LIN {X 0,Y 579.036,Z 911.007,A -85,B 0,C 180,E1 18401.072,E2 18401.072} C_VEL
LIN {X 0,Y 580.6,Z 886.113,A -85,B 0,C 180,E1 18400.644,E2 18400.644} C_VEL
LIN {X 0,Y 588.894,Z 664.984,A -85,B 0,C 180,E1 18397.408,E2 18397.408} C_VEL
LIN {X 0,Y 594.592,Z 519.024,A -85,B 0,C 180,E1 18395.226,E2 18395.226} C_VEL
LIN {X 0,Y 583.238,Z 502.183,A -85,B 0,C 180,E1 18393.242,E2 18393.242} C_VEL
LIN {X 0,Y 573.346,Z 488.224,A -85,B 0,C 180,E1 18391.371,E2 18391.371} C_VEL
LIN {X 0,Y 562.808,Z 474.786,A -85,B 0,C 180,E1 18389.217,E2 18389.217} C_VEL
LIN {X 0,Y 557.617,Z 468.552,A -85,B 0,C 180,E1 18388.08,E2 18388.08} C_VEL
LIN {X 0,Y 553.132,Z 463.086,A -85,B 0,C 180,E1 18387.042,E2 18387.042} C_VEL
LIN {X 0,Y 548.609,Z 457.659,A -85,B 0,C 180,E1 18385.94,E2 18385.94} C_VEL
LIN {X 0,Y 544.992,Z 453.494,A -85,B 0,C 180,E1 18385.018,E2 18385.018} C_VEL
LIN {X 0,Y 543.71,Z 451.828,A -85,B 0,C 180,E1 18384.674,E2 18384.674} C_VEL
LIN {X 0,Y 540.306,Z 448.41,A -85,B 0,C 180,E1 18383.764,E2 18383.764} C_VEL
LIN {X 0,Y 538.516,Z 445.758,A -85,B 0,C 180,E1 18383.239,E2 18383.239} C_VEL
LIN {X 0,Y 535.176,Z 442.868,A -85,B 0,C 180,E1 18382.289,E2 18382.289} C_VEL
LIN {X 0,Y 532.967,Z 439.362,A -85,B 0,C 180,E1 18381.575,E2 18381.575} C_VEL
LIN {X 0,Y 529.819,Z 437.07,A -85,B 0,C 180,E1 18380.608,E2 18380.608} C_VEL
LIN {X 0,Y 527.865,Z 433.796,A -85,B 0,C 180,E1 18379.907,E2 18379.907} C_VEL
LIN {X 0,Y 527.382,Z 432.859,A -85,B 0,C 180,E1 18379.723,E2 18379.723} C_VEL
LIN {X 0,Y 524.15,Z 431.063,A -85,B 0,C 180,E1 18378.635,E2 18378.635} C_VEL
LIN {X 0,Y 522.344,Z 428.45,A -85,B 0,C 180,E1 18377.922,E2 18377.922} C_VEL
LIN {X 0,Y 521.734,Z 426.245,A -85,B 0,C 180,E1 18377.569,E2 18377.569} C_VEL
LIN {X 0,Y 521.677,Z 426.183,A -85,B 0,C 180,E1 18374.315,E2 18374.315} C_VEL
LIN {X 0,Y 521.681,Z 426.216,A -85,B 0,C 180,E1 18370.826,E2 18370.826} C_VEL
LIN {X 0,Y 521.736,Z 426.191,A -85,B 0,C 180,E1 18367.488,E2 18367.488} C_VEL
LIN {X 0,Y 521.667,Z 426.198,A -85,B 0,C 180,E1 18364.177,E2 18364.177} C_VEL
LIN {X 0,Y 521.698,Z 426.217,A -85,B 0,C 180,E1 18360.769,E2 18360.769} C_VEL
LIN {X 0,Y 521.675,Z 426.189,A -85,B 0,C 180,E1 18357.693,E2 18357.693} C_VEL
LIN {X 0,Y 521.674,Z 426.24,A -85,B 0,C 180,E1 18354.17,E2 18354.17} C_VEL
LIN {X 0,Y 521.705,Z 426.178,A -85,B 0,C 180,E1 18351.069,E2 18351.069} C_VEL
LIN {X 0,Y 521.667,Z 426.25,A -85,B 0,C 180,E1 18347.716,E2 18347.716} C_VEL
LIN {X 0,Y 521.718,Z 426.177,A -85,B 0,C 180,E1 18344.436,E2 18344.436} C_VEL
LIN {X 0,Y 521.761,Z 426.459,A -85,B 0,C 180,E1 18342.476,E2 18342.476} C_VEL
LIN {X 0,Y 522.696,Z 429.249,A -85,B 0,C 180,E1 18342.033,E2 18342.033} C_VEL
LIN {X 0,Y 525.013,Z 431.775,A -85,B 0,C 180,E1 18341.167,E2 18341.167} C_VEL
LIN {X 0,Y 527.588,Z 433.099,A -85,B 0,C 180,E1 18340.313,E2 18340.313} C_VEL
LIN {X 0,Y 529.339,Z 436.508,A -85,B 0,C 180,E1 18339.661,E2 18339.661} C_VEL
LIN {X 0,Y 532.257,Z 439.002,A -85,B 0,C 180,E1 18338.742,E2 18338.742} C_VEL
LIN {X 0,Y 533.358,Z 439.775,A -85,B 0,C 180,E1 18338.413,E2 18338.413} C_VEL
LIN {X 0,Y 535.655,Z 443.463,A -85,B 0,C 180,E1 18337.674,E2 18337.674} C_VEL
LIN {X 0,Y 539.017,Z 446.356,A -85,B 0,C 180,E1 18336.726,E2 18336.726} C_VEL
LIN {X 0,Y 541.984,Z 450.42,A -85,B 0,C 180,E1 18335.881,E2 18335.881} C_VEL
LIN {X 0,Y 544.316,Z 452.723,A -85,B 0,C 180,E1 18335.268,E2 18335.268} C_VEL
LIN {X 0,Y 552.544,Z 463.032,A -85,B 0,C 180,E1 18333.189,E2 18333.189} C_VEL
LIN {X 0,Y 558.316,Z 470.524,A -85,B 0,C 180,E1 18331.842,E2 18331.842} C_VEL
LIN {X 0,Y 566.802,Z 481.647,A -85,B 0,C 180,E1 18330.006,E2 18330.006} C_VEL
LIN {X 0,Y 579.311,Z 499.123,A -85,B 0,C 180,E1 18327.535,E2 18327.535} C_VEL
LIN {X 0,Y 591.797,Z 517.896,A -85,B 0,C 180,E1 18325.292,E2 18325.292} C_VEL
LIN {X 0,Y 594.718,Z 522.57,A -85,B 0,C 180,E1 18324.793,E2 18324.793} C_VEL
LIN {X 0,Y 586.211,Z 739.964,A -85,B 0,C 180,E1 18321.576,E2 18321.576} C_VEL
LIN {X 0,Y 580.04,Z 903.137,A -85,B 0,C 180,E1 18319.182,E2 18319.182} C_VEL
LIN {X 0,Y 578.241,Z 928.181,A -85,B 0,C 180,E1 18318.717,E2 18318.717} C_VEL
LIN {X 0,Y 575.436,Z 956.17,A -85,B 0,C 180,E1 18318.007,E2 18318.007} C_VEL
LIN {X 0,Y 572.745,Z 978.261,A -85,B 0,C 180,E1 18317.298,E2 18317.298} C_VEL
LIN {X 0,Y 569.876,Z 998.966,A -85,B 0,C 180,E1 18316.505,E2 18316.505} C_VEL
LIN {X 0,Y 566.742,Z 1019.265,A -85,B 0,C 180,E1 18315.598,E2 18315.598} C_VEL
LIN {X 0,Y 562.552,Z 1044.182,A -85,B 0,C 180,E1 18314.302,E2 18314.302} C_VEL
LIN {X 0,Y 558.22,Z 1067.089,A -85,B 0,C 180,E1 18312.889,E2 18312.889} C_VEL
LIN {X 0,Y 554.385,Z 1086.314,A -85,B 0,C 180,E1 18311.539,E2 18311.539} C_VEL
LIN {X 0,Y 550.54,Z 1104.879,A -85,B 0,C 180,E1 18310.073,E2 18310.073} C_VEL
LIN {X 0,Y 546.407,Z 1124.422,A -85,B 0,C 180,E1 18308.335,E2 18308.335} C_VEL
LIN {X 0,Y 541.6,Z 1146.573,A -85,B 0,C 180,E1 18306.075,E2 18306.075} C_VEL
LIN {X 0,Y 538.12,Z 1162.602,A -85,B 0,C 180,E1 18304.222,E2 18304.222} C_VEL
LIN {X 0,Y 534.941,Z 1177.486,A -85,B 0,C 180,E1 18302.31,E2 18302.31} C_VEL
LIN {X 0,Y 532.102,Z 1191.164,A -85,B 0,C 180,E1 18300.358,E2 18300.358} C_VEL
LIN {X 0,Y 528.99,Z 1207.163,A -85,B 0,C 180,E1 18297.796,E2 18297.796} C_VEL
LIN {X 0,Y 526.229,Z 1221.856,A -85,B 0,C 180,E1 18295.065,E2 18295.065} C_VEL
LIN {X 0,Y 524.427,Z 1232.786,A -85,B 0,C 180,E1 18292.766,E2 18292.766} C_VEL
LIN {X 0,Y 522.967,Z 1242.909,A -85,B 0,C 180,E1 18290.359,E2 18290.359} C_VEL
LIN {X 0,Y 521.584,Z 1254.042,A -85,B 0,C 180,E1 18287.282,E2 18287.282} C_VEL
LIN {X 0,Y 520.803,Z 1261.844,A -85,B 0,C 180,E1 18284.676,E2 18284.676} C_VEL
LIN {X 0,Y 520.369,Z 1267.807,A -85,B 0,C 180,E1 18282.311,E2 18282.311} C_VEL
LIN {X 0,Y 520.093,Z 1272.702,A -85,B 0,C 180,E1 18279.96,E2 18279.96} C_VEL
LIN {X 0,Y 519.964,Z 1276.525,A -85,B 0,C 180,E1 18277.621,E2 18277.621} C_VEL
LIN {X 0,Y 519.925,Z 1279.433,A -85,B 0,C 180,E1 18275.182,E2 18275.182} C_VEL
LIN {X 0,Y 519.907,Z 1281.491,A -85,B 0,C 180,E1 18272.311,E2 18272.311} C_VEL
LIN {X 0,Y 519.867,Z 1281.893,A -85,B 0,C 180,E1 18269.446,E2 18269.446} C_VEL
LIN {X 0,Y 519.91,Z 1281.08,A -85,B 0,C 180,E1 18267.02,E2 18267.02} C_VEL
LIN {X 0,Y 519.926,Z 1279.198,A -85,B 0,C 180,E1 18264.59,E2 18264.59} C_VEL
LIN {X 0,Y 519.965,Z 1276.355,A -85,B 0,C 180,E1 18262.261,E2 18262.261} C_VEL
LIN {X 0,Y 520.127,Z 1272.277,A -85,B 0,C 180,E1 18259.81,E2 18259.81} C_VEL
LIN {X 0,Y 520.467,Z 1266.52,A -85,B 0,C 180,E1 18257.121,E2 18257.121} C_VEL
LIN {X 0,Y 521.149,Z 1258.259,A -85,B 0,C 180,E1 18254.073,E2 18254.073} C_VEL
LIN {X 0,Y 522.037,Z 1250.093,A -85,B 0,C 180,E1 18251.574,E2 18251.574} C_VEL
LIN {X 0,Y 523.226,Z 1241.051,A -85,B 0,C 180,E1 18249.177,E2 18249.177} C_VEL
LIN {X 0,Y 524.865,Z 1230.188,A -85,B 0,C 180,E1 18246.654,E2 18246.654} C_VEL
LIN {X 0,Y 527.442,Z 1215.245,A -85,B 0,C 180,E1 18243.664,E2 18243.664} C_VEL
LIN {X 0,Y 529.901,Z 1202.05,A -85,B 0,C 180,E1 18241.359,E2 18241.359} C_VEL
LIN {X 0,Y 532.597,Z 1188.807,A -85,B 0,C 180,E1 18239.291,E2 18239.291} C_VEL
LIN {X 0,Y 535.704,Z 1174.039,A -85,B 0,C 180,E1 18237.227,E2 18237.227} C_VEL
LIN {X 0,Y 540.173,Z 1153.102,A -85,B 0,C 180,E1 18234.652,E2 18234.652} C_VEL
LIN {X 0,Y 543.91,Z 1135.76,A -85,B 0,C 180,E1 18232.783,E2 18232.783} C_VEL
LIN {X 0,Y 547.556,Z 1118.85,A -85,B 0,C 180,E1 18231.15,E2 18231.15} C_VEL
LIN {X 0,Y 551.544,Z 1100.101,A -85,B 0,C 180,E1 18229.531,E2 18229.531} C_VEL
LIN {X 0,Y 556.662,Z 1075.128,A -85,B 0,C 180,E1 18227.654,E2 18227.654} C_VEL
LIN {X 0,Y 560.526,Z 1054.925,A -85,B 0,C 180,E1 18226.341,E2 18226.341} C_VEL
LIN {X 0,Y 563.912,Z 1036.027,A -85,B 0,C 180,E1 18225.255,E2 18225.255} C_VEL
LIN {X 0,Y 567.295,Z 1015.734,A -85,B 0,C 180,E1 18224.234,E2 18224.234} C_VEL
LIN {X 0,Y 570.571,Z 994.236,A -85,B 0,C 180,E1 18223.301,E2 18223.301} C_VEL
LIN {X 0,Y 574.261,Z 966.352,A -85,B 0,C 180,E1 18222.3,E2 18222.3} C_VEL
LIN {X 0,Y 576.846,Z 942.712,A -85,B 0,C 180,E1 18221.629,E2 18221.629} C_VEL
LIN {X 0,Y 578.774,Z 921.217,A -85,B 0,C 180,E1 18221.143,E2 18221.143} C_VEL
LIN {X 0,Y 580.258,Z 898.846,A -85,B 0,C 180,E1 18220.75,E2 18220.75} C_VEL
LIN {X 0,Y 588.488,Z 679.578,A -85,B 0,C 180,E1 18217.538,E2 18217.538} C_VEL
LIN {X 0,Y 594.641,Z 522.279,A -85,B 0,C 180,E1 18215.196,E2 18215.196} C_VEL
LIN {X 0,Y 582.085,Z 503.302,A -85,B 0,C 180,E1 18212.993,E2 18212.993} C_VEL
LIN {X 0,Y 571.124,Z 487.581,A -85,B 0,C 180,E1 18210.891,E2 18210.891} C_VEL
LIN {X 0,Y 559.93,Z 472.501,A -85,B 0,C 180,E1 18208.535,E2 18208.535} C_VEL
LIN {X 0,Y 554.757,Z 466.005,A -85,B 0,C 180,E1 18207.362,E2 18207.362} C_VEL
LIN {X 0,Y 550.787,Z 460.835,A -85,B 0,C 180,E1 18206.409,E2 18206.409} C_VEL
LIN {X 0,Y 543.204,Z 451.467,A -85,B 0,C 180,E1 18204.467,E2 18204.467} C_VEL
LIN {X 0,Y 539.929,Z 447.877,A -85,B 0,C 180,E1 18203.579,E2 18203.579} C_VEL
LIN {X 0,Y 538.57,Z 445.796,A -85,B 0,C 180,E1 18203.178,E2 18203.178} C_VEL
LIN {X 0,Y 535.297,Z 443.031,A -85,B 0,C 180,E1 18202.255,E2 18202.255} C_VEL
LIN {X 0,Y 533.175,Z 439.455,A -85,B 0,C 180,E1 18201.566,E2 18201.566} C_VEL
LIN {X 0,Y 529.837,Z 437.087,A -85,B 0,C 180,E1 18200.549,E2 18200.549} C_VEL
LIN {X 0,Y 527.874,Z 433.805,A -85,B 0,C 180,E1 18199.848,E2 18199.848} C_VEL
LIN {X 0,Y 527.553,Z 432.909,A -85,B 0,C 180,E1 18199.717,E2 18199.717} C_VEL
LIN {X 0,Y 524.143,Z 431.05,A -85,B 0,C 180,E1 18198.577,E2 18198.577} C_VEL
LIN {X 0,Y 522.271,Z 428.25,A -85,B 0,C 180,E1 18197.838,E2 18197.838} C_VEL
LIN {X 0,Y 521.734,Z 426.244,A -85,B 0,C 180,E1 18197.54,E2 18197.54} C_VEL
LIN {X 0,Y 521.706,Z 426.183,A -85,B 0,C 180,E1 18194.201,E2 18194.201} C_VEL
LIN {X 0,Y 521.699,Z 426.209,A -85,B 0,C 180,E1 18190.826,E2 18190.826} C_VEL
LIN {X 0,Y 521.751,Z 426.198,A -85,B 0,C 180,E1 18187.377,E2 18187.377} C_VEL
LIN {X 0,Y 521.711,Z 426.185,A -85,B 0,C 180,E1 18184.066,E2 18184.066} C_VEL
LIN {X 0,Y 521.713,Z 426.233,A -85,B 0,C 180,E1 18180.549,E2 18180.549} C_VEL
LIN {X 0,Y 521.737,Z 426.171,A -85,B 0,C 180,E1 18177.144,E2 18177.144} C_VEL
LIN {X 0,Y 521.743,Z 426.239,A -85,B 0,C 180,E1 18173.618,E2 18173.618} C_VEL
LIN {X 0,Y 521.718,Z 426.181,A -85,B 0,C 180,E1 18170.099,E2 18170.099} C_VEL
LIN {X 0,Y 521.743,Z 426.202,A -85,B 0,C 180,E1 18166.704,E2 18166.704} C_VEL
LIN {X 0,Y 521.738,Z 426.209,A -85,B 0,C 180,E1 18163.179,E2 18163.179} C_VEL
LIN {X 0,Y 521.765,Z 426.425,A -85,B 0,C 180,E1 18162.216,E2 18162.216} C_VEL
LIN {X 0,Y 522.647,Z 429.071,A -85,B 0,C 180,E1 18161.801,E2 18161.801} C_VEL
LIN {X 0,Y 525.115,Z 431.787,A -85,B 0,C 180,E1 18160.882,E2 18160.882} C_VEL
LIN {X 0,Y 527.676,Z 433.195,A -85,B 0,C 180,E1 18160.036,E2 18160.036} C_VEL
LIN {X 0,Y 529.467,Z 436.573,A -85,B 0,C 180,E1 18159.378,E2 18159.378} C_VEL
LIN {X 0,Y 532.576,Z 439.16,A -85,B 0,C 180,E1 18158.409,E2 18158.409} C_VEL
LIN {X 0,Y 533.5,Z 439.944,A -85,B 0,C 180,E1 18158.13,E2 18158.13} C_VEL
LIN {X 0,Y 535.819,Z 443.573,A -85,B 0,C 180,E1 18157.392,E2 18157.392} C_VEL
LIN {X 0,Y 539.108,Z 446.411,A -85,B 0,C 180,E1 18156.47,E2 18156.47} C_VEL
LIN {X 0,Y 541.999,Z 450.36,A -85,B 0,C 180,E1 18155.649,E2 18155.649} C_VEL
LIN {X 0,Y 544.45,Z 452.616,A -85,B 0,C 180,E1 18155.014,E2 18155.014} C_VEL
LIN {X 0,Y 547.821,Z 456.922,A -85,B 0,C 180,E1 18154.137,E2 18154.137} C_VEL
LIN {X 0,Y 549.689,Z 458.859,A -85,B 0,C 180,E1 18153.68,E2 18153.68} C_VEL
LIN {X 0,Y 553.558,Z 463.505,A -85,B 0,C 180,E1 18152.748,E2 18152.748} C_VEL
LIN {X 0,Y 559.954,Z 471.36,A -85,B 0,C 180,E1 18151.292,E2 18151.292} C_VEL
LIN {X 0,Y 568.098,Z 481.467,A -85,B 0,C 180,E1 18149.572,E2 18149.572} C_VEL
LIN {X 0,Y 576.042,Z 491.922,A -85,B 0,C 180,E1 18148.004,E2 18148.004} C_VEL
LIN {X 0,Y 588.387,Z 509.679,A -85,B 0,C 180,E1 18145.742,E2 18145.742} C_VEL
LIN {X 0,Y 594.647,Z 519.437,A -85,B 0,C 180,E1 18144.662,E2 18144.662} C_VEL
LIN {X 0,Y 586.266,Z 733.251,A -85,B 0,C 180,E1 18141.497,E2 18141.497} C_VEL
LIN {X 0,Y 580.128,Z 894.828,A -85,B 0,C 180,E1 18139.126,E2 18139.126} C_VEL
LIN {X 0,Y 578.382,Z 919.425,A -85,B 0,C 180,E1 18138.667,E2 18138.667} C_VEL
LIN {X 0,Y 575.597,Z 947.533,A -85,B 0,C 180,E1 18137.952,E2 18137.952} C_VEL
LIN {X 0,Y 573.377,Z 966.175,A -85,B 0,C 180,E1 18137.362,E2 18137.362} C_VEL
LIN {X 0,Y 571.693,Z 973.633,A -85,B 0,C 180,E1 18137.174,E2 18137.174} C_VEL
LIN {X 0,Y 564.929,Z 992.335,A -85,B 0,C 180,E1 18136.894,E2 18136.894} C_VEL
LIN {X 0,Y 563.145,Z 999.439,A -85,B 0,C 180,E1 18136.66,E2 18136.66} C_VEL
LIN {X 0,Y 558.919,Z 1024.068,A -85,B 0,C 180,E1 18135.448,E2 18135.448} C_VEL
LIN {X 0,Y 555.437,Z 1042.82,A -85,B 0,C 180,E1 18134.383,E2 18134.383} C_VEL
LIN {X 0,Y 551.84,Z 1060.85,A -85,B 0,C 180,E1 18133.23,E2 18133.23} C_VEL
LIN {X 0,Y 547.962,Z 1079.276,A -85,B 0,C 180,E1 18131.903,E2 18131.903} C_VEL
LIN {X 0,Y 543.746,Z 1098.556,A -85,B 0,C 180,E1 18130.339,E2 18130.339} C_VEL
LIN {X 0,Y 538.534,Z 1121.584,A -85,B 0,C 180,E1 18128.192,E2 18128.192} C_VEL
LIN {X 0,Y 534.458,Z 1139.111,A -85,B 0,C 180,E1 18126.322,E2 18126.322} C_VEL
LIN {X 0,Y 530.92,Z 1154.438,A -85,B 0,C 180,E1 18124.496,E2 18124.496} C_VEL
LIN {X 0,Y 527.405,Z 1169.864,A -85,B 0,C 180,E1 18122.45,E2 18122.45} C_VEL
LIN {X 0,Y 523.546,Z 1187.627,A -85,B 0,C 180,E1 18119.775,E2 18119.775} C_VEL
LIN {X 0,Y 520.587,Z 1201.836,A -85,B 0,C 180,E1 18117.328,E2 18117.328} C_VEL
LIN {X 0,Y 518.387,Z 1213.335,A -85,B 0,C 180,E1 18115.111,E2 18115.111} C_VEL
LIN {X 0,Y 516.527,Z 1224.112,A -85,B 0,C 180,E1 18112.78,E2 18112.78} C_VEL
LIN {X 0,Y 514.77,Z 1235.881,A -85,B 0,C 180,E1 18109.874,E2 18109.874} C_VEL
LIN {X 0,Y 513.521,Z 1245.65,A -85,B 0,C 180,E1 18106.984,E2 18106.984} C_VEL
LIN {X 0,Y 512.833,Z 1252.312,A -85,B 0,C 180,E1 18104.685,E2 18104.685} C_VEL
LIN {X 0,Y 512.394,Z 1257.946,A -85,B 0,C 180,E1 18102.398,E2 18102.398} C_VEL
LIN {X 0,Y 512.109,Z 1262.812,A -85,B 0,C 180,E1 18100.01,E2 18100.01} C_VEL
LIN {X 0,Y 511.962,Z 1266.768,A -85,B 0,C 180,E1 18097.522,E2 18097.522} C_VEL
LIN {X 0,Y 511.921,Z 1269.832,A -85,B 0,C 180,E1 18094.821,E2 18094.821} C_VEL
LIN {X 0,Y 511.908,Z 1271.634,A -85,B 0,C 180,E1 18091.794,E2 18091.794} C_VEL
LIN {X 0,Y 511.865,Z 1271.858,A -85,B 0,C 180,E1 18089.22,E2 18089.22} C_VEL
LIN {X 0,Y 511.911,Z 1271.043,A -85,B 0,C 180,E1 18086.868,E2 18086.868} C_VEL
LIN {X 0,Y 511.928,Z 1269.249,A -85,B 0,C 180,E1 18084.512,E2 18084.512} C_VEL
LIN {X 0,Y 511.973,Z 1266.426,A -85,B 0,C 180,E1 18082.146,E2 18082.146} C_VEL
LIN {X 0,Y 512.147,Z 1262.368,A -85,B 0,C 180,E1 18079.656,E2 18079.656} C_VEL
LIN {X 0,Y 512.511,Z 1256.635,A -85,B 0,C 180,E1 18076.924,E2 18076.924} C_VEL
LIN {X 0,Y 513.225,Z 1248.418,A -85,B 0,C 180,E1 18073.828,E2 18073.828} C_VEL
LIN {X 0,Y 514.17,Z 1240.216,A -85,B 0,C 180,E1 18071.273,E2 18071.273} C_VEL
LIN {X 0,Y 515.427,Z 1231.245,A -85,B 0,C 180,E1 18068.854,E2 18068.854} C_VEL
LIN {X 0,Y 517.076,Z 1220.916,A -85,B 0,C 180,E1 18066.409,E2 18066.409} C_VEL
LIN {X 0,Y 519.684,Z 1206.642,A -85,B 0,C 180,E1 18063.467,E2 18063.467} C_VEL
LIN {X 0,Y 522.37,Z 1192.914,A -85,B 0,C 180,E1 18061.018,E2 18061.018} C_VEL
LIN {X 0,Y 525.169,Z 1179.971,A -85,B 0,C 180,E1 18058.943,E2 18058.943} C_VEL
LIN {X 0,Y 528.229,Z 1166.296,A -85,B 0,C 180,E1 18056.97,E2 18056.97} C_VEL
LIN {X 0,Y 531.991,Z 1149.884,A -85,B 0,C 180,E1 18054.845,E2 18054.845} C_VEL
LIN {X 0,Y 536.787,Z 1129.016,A -85,B 0,C 180,E1 18052.481,E2 18052.481} C_VEL
LIN {X 0,Y 540.792,Z 1111.502,A -85,B 0,C 180,E1 18050.739,E2 18050.739} C_VEL
LIN {X 0,Y 544.691,Z 1094.186,A -85,B 0,C 180,E1 18049.2,E2 18049.2} C_VEL
LIN {X 0,Y 548.793,Z 1075.37,A -85,B 0,C 180,E1 18047.708,E2 18047.708} C_VEL
LIN {X 0,Y 553.8,Z 1051.295,A -85,B 0,C 180,E1 18046.042,E2 18046.042} C_VEL
LIN {X 0,Y 557.992,Z 1029.086,A -85,B 0,C 180,E1 18044.731,E2 18044.731} C_VEL
LIN {X 0,Y 561.497,Z 1009.094,A -85,B 0,C 180,E1 18043.704,E2 18043.704} C_VEL
LIN {X 0,Y 564.561,Z 989.967,A -85,B 0,C 180,E1 18042.849,E2 18042.849} C_VEL
LIN {X 0,Y 567.434,Z 969.925,A -85,B 0,C 180,E1 18042.076,E2 18042.076} C_VEL
LIN {X 0,Y 570.195,Z 947.979,A -85,B 0,C 180,E1 18041.366,E2 18041.366} C_VEL
LIN {X 0,Y 573.055,Z 920.319,A -85,B 0,C 180,E1 18040.655,E2 18040.655} C_VEL
LIN {X 0,Y 574.916,Z 895.077,A -85,B 0,C 180,E1 18040.181,E2 18040.181} C_VEL
LIN {X 0,Y 580.74,Z 748.236,A -85,B 0,C 180,E1 18038.012,E2 18038.012} C_VEL
LIN {X 0,Y 589.427,Z 534.986,A -85,B 0,C 180,E1 18034.843,E2 18034.843} C_VEL
LIN {X 0,Y 589.825,Z 523.275,A -85,B 0,C 180,E1 18034.653,E2 18034.653} C_VEL
LIN {X 0,Y 579.401,Z 507.75,A -85,B 0,C 180,E1 18032.782,E2 18032.782} C_VEL
LIN {X 0,Y 569.991,Z 494.34,A -85,B 0,C 180,E1 18030.959,E2 18030.959} C_VEL
LIN {X 0,Y 559.803,Z 481.353,A -85,B 0,C 180,E1 18028.833,E2 18028.833} C_VEL
LIN {X 0,Y 554.789,Z 475.248,A -85,B 0,C 180,E1 18027.71,E2 18027.71} C_VEL
LIN {X 0,Y 550.666,Z 470.149,A -85,B 0,C 180,E1 18026.735,E2 18026.735} C_VEL
LIN {X 0,Y 546.293,Z 464.859,A -85,B 0,C 180,E1 18025.65,E2 18025.65} C_VEL
LIN {X 0,Y 542.548,Z 460.371,A -85,B 0,C 180,E1 18024.672,E2 18024.672} C_VEL
LIN {X 0,Y 541.071,Z 458.796,A -85,B 0,C 180,E1 18024.279,E2 18024.279} C_VEL
LIN {X 0,Y 537.596,Z 454.789,A -85,B 0,C 180,E1 18023.31,E2 18023.31} C_VEL
LIN {X 0,Y 536.497,Z 453.235,A -85,B 0,C 180,E1 18022.983,E2 18022.983} C_VEL
LIN {X 0,Y 533.047,Z 450.017,A -85,B 0,C 180,E1 18021.976,E2 18021.976} C_VEL
LIN {X 0,Y 531.01,Z 446.911,A -85,B 0,C 180,E1 18021.31,E2 18021.31} C_VEL
LIN {X 0,Y 527.773,Z 444.256,A -85,B 0,C 180,E1 18020.286,E2 18020.286} C_VEL
LIN {X 0,Y 525.492,Z 440.526,A -85,B 0,C 180,E1 18019.45,E2 18019.45} C_VEL
LIN {X 0,Y 522.199,Z 438.327,A -85,B 0,C 180,E1 18018.302,E2 18018.302} C_VEL
LIN {X 0,Y 520.267,Z 435.183,A -85,B 0,C 180,E1 18017.504,E2 18017.504} C_VEL
LIN {X 0,Y 519.808,Z 434.015,A -85,B 0,C 180,E1 18017.289,E2 18017.289} C_VEL
LIN {X 0,Y 516.455,Z 432.216,A -85,B 0,C 180,E1 18015.957,E2 18015.957} C_VEL
LIN {X 0,Y 514.286,Z 429.246,A -85,B 0,C 180,E1 18014.928,E2 18014.928} C_VEL
LIN {X 0,Y 513.731,Z 427.169,A -85,B 0,C 180,E1 18014.541,E2 18014.541} C_VEL
LIN {X 0,Y 513.765,Z 427.211,A -85,B 0,C 180,E1 18011.109,E2 18011.109} C_VEL
LIN {X 0,Y 513.757,Z 427.174,A -85,B 0,C 180,E1 18007.83,E2 18007.83} C_VEL
LIN {X 0,Y 513.733,Z 427.192,A -85,B 0,C 180,E1 18004.465,E2 18004.465} C_VEL
LIN {X 0,Y 513.796,Z 427.185,A -85,B 0,C 180,E1 18001.115,E2 18001.115} C_VEL
LIN {X 0,Y 513.728,Z 427.18,A -85,B 0,C 180,E1 17997.881,E2 17997.881} C_VEL
LIN {X 0,Y 513.748,Z 427.214,A -85,B 0,C 180,E1 17994.415,E2 17994.415} C_VEL
LIN {X 0,Y 513.742,Z 427.17,A -85,B 0,C 180,E1 17991.344,E2 17991.344} C_VEL
LIN {X 0,Y 513.731,Z 427.239,A -85,B 0,C 180,E1 17987.866,E2 17987.866} C_VEL
LIN {X 0,Y 513.739,Z 427.322,A -85,B 0,C 180,E1 17985.517,E2 17985.517} C_VEL
LIN {X 0,Y 514.585,Z 429.867,A -85,B 0,C 180,E1 17985.023,E2 17985.023} C_VEL
LIN {X 0,Y 517.197,Z 432.829,A -85,B 0,C 180,E1 17983.836,E2 17983.836} C_VEL
LIN {X 0,Y 519.913,Z 434.245,A -85,B 0,C 180,E1 17982.772,E2 17982.772} C_VEL
LIN {X 0,Y 521.498,Z 437.521,A -85,B 0,C 180,E1 17982.077,E2 17982.077} C_VEL
LIN {X 0,Y 524.383,Z 440.031,A -85,B 0,C 180,E1 17981.026,E2 17981.026} C_VEL
LIN {X 0,Y 525.766,Z 440.869,A -85,B 0,C 180,E1 17980.56,E2 17980.56} C_VEL
LIN {X 0,Y 527.906,Z 444.43,A -85,B 0,C 180,E1 17979.777,E2 17979.777} C_VEL
LIN {X 0,Y 531.473,Z 447.447,A -85,B 0,C 180,E1 17978.651,E2 17978.651} C_VEL
LIN {X 0,Y 534.186,Z 451.376,A -85,B 0,C 180,E1 17977.784,E2 17977.784} C_VEL
LIN {X 0,Y 536.992,Z 453.833,A -85,B 0,C 180,E1 17976.982,E2 17976.982} C_VEL
LIN {X 0,Y 540.118,Z 457.965,A -85,B 0,C 180,E1 17976.082,E2 17976.082} C_VEL
LIN {X 0,Y 542.512,Z 460.465,A -85,B 0,C 180,E1 17975.442,E2 17975.442} C_VEL
LIN {X 0,Y 550.279,Z 470.345,A -85,B 0,C 180,E1 17973.449,E2 17973.449} C_VEL
LIN {X 0,Y 558.284,Z 480.701,A -85,B 0,C 180,E1 17971.578,E2 17971.578} C_VEL
LIN {X 0,Y 569.062,Z 495.522,A -85,B 0,C 180,E1 17969.278,E2 17969.278} C_VEL
LIN {X 0,Y 579.122,Z 510.073,A -85,B 0,C 180,E1 17967.317,E2 17967.317} C_VEL
LIN {X 0,Y 589.944,Z 526.608,A -85,B 0,C 180,E1 17965.369,E2 17965.369} C_VEL
LIN {X 0,Y 581.1,Z 743.647,A -85,B 0,C 180,E1 17962.142,E2 17962.142} C_VEL
LIN {X 0,Y 574.825,Z 902.956,A -85,B 0,C 180,E1 17959.79,E2 17959.79} C_VEL
LIN {X 0,Y 572.972,Z 927.943,A -85,B 0,C 180,E1 17959.326,E2 17959.326} C_VEL
LIN {X 0,Y 570.058,Z 956.08,A -85,B 0,C 180,E1 17958.611,E2 17958.611} C_VEL
LIN {X 0,Y 567.273,Z 978.178,A -85,B 0,C 180,E1 17957.9,E2 17957.9} C_VEL
LIN {X 0,Y 564.321,Z 998.754,A -85,B 0,C 180,E1 17957.11,E2 17957.11} C_VEL
LIN {X 0,Y 561.042,Z 1019.18,A -85,B 0,C 180,E1 17956.195,E2 17956.195} C_VEL
LIN {X 0,Y 556.686,Z 1044.095,A -85,B 0,C 180,E1 17954.894,E2 17954.894} C_VEL
LIN {X 0,Y 552.016,Z 1067.808,A -85,B 0,C 180,E1 17953.419,E2 17953.419} C_VEL
LIN {X 0,Y 547.988,Z 1087.181,A -85,B 0,C 180,E1 17952.043,E2 17952.043} C_VEL
LIN {X 0,Y 544.037,Z 1105.458,A -85,B 0,C 180,E1 17950.582,E2 17950.582} C_VEL
LIN {X 0,Y 539.227,Z 1127.368,A -85,B 0,C 180,E1 17948.601,E2 17948.601} C_VEL
LIN {X 0,Y 534.599,Z 1147.5,A -85,B 0,C 180,E1 17946.491,E2 17946.491} C_VEL
LIN {X 0,Y 530.982,Z 1163.398,A -85,B 0,C 180,E1 17944.622,E2 17944.622} C_VEL
LIN {X 0,Y 527.663,Z 1178.244,A -85,B 0,C 180,E1 17942.682,E2 17942.682} C_VEL
LIN {X 0,Y 524.012,Z 1195.317,A -85,B 0,C 180,E1 17940.186,E2 17940.186} C_VEL
LIN {X 0,Y 520.791,Z 1210.83,A -85,B 0,C 180,E1 17937.557,E2 17937.557} C_VEL
LIN {X 0,Y 518.462,Z 1222.903,A -85,B 0,C 180,E1 17935.243,E2 17935.243} C_VEL
LIN {X 0,Y 516.662,Z 1233.298,A -85,B 0,C 180,E1 17933.008,E2 17933.008} C_VEL
LIN {X 0,Y 514.998,Z 1244.284,A -85,B 0,C 180,E1 17930.332,E2 17930.332} C_VEL
LIN {X 0,Y 513.582,Z 1255.103,A -85,B 0,C 180,E1 17927.209,E2 17927.209} C_VEL
LIN {X 0,Y 512.836,Z 1262.276,A -85,B 0,C 180,E1 17924.745,E2 17924.745} C_VEL
LIN {X 0,Y 512.389,Z 1268.061,A -85,B 0,C 180,E1 17922.391,E2 17922.391} C_VEL
LIN {X 0,Y 512.102,Z 1272.906,A -85,B 0,C 180,E1 17920.004,E2 17920.004} C_VEL
LIN {X 0,Y 511.967,Z 1276.842,A -85,B 0,C 180,E1 17917.515,E2 17917.515} C_VEL
LIN {X 0,Y 511.92,Z 1279.996,A -85,B 0,C 180,E1 17914.702,E2 17914.702} C_VEL
LIN {X 0,Y 511.908,Z 1281.668,A -85,B 0,C 180,E1 17911.676,E2 17911.676} C_VEL
LIN {X 0,Y 511.866,Z 1281.848,A -85,B 0,C 180,E1 17909.213,E2 17909.213} C_VEL
LIN {X 0,Y 511.91,Z 1281.012,A -85,B 0,C 180,E1 17906.862,E2 17906.862} C_VEL
LIN {X 0,Y 511.929,Z 1279.196,A -85,B 0,C 180,E1 17904.505,E2 17904.505} C_VEL
LIN {X 0,Y 511.972,Z 1276.352,A -85,B 0,C 180,E1 17902.14,E2 17902.14} C_VEL
LIN {X 0,Y 512.156,Z 1272.274,A -85,B 0,C 180,E1 17899.65,E2 17899.65} C_VEL
LIN {X 0,Y 512.552,Z 1266.189,A -85,B 0,C 180,E1 17896.77,E2 17896.77} C_VEL
LIN {X 0,Y 513.279,Z 1257.905,A -85,B 0,C 180,E1 17893.706,E2 17893.706} C_VEL
LIN {X 0,Y 514.228,Z 1249.687,A -85,B 0,C 180,E1 17891.167,E2 17891.167} C_VEL
LIN {X 0,Y 515.457,Z 1241.049,A -85,B 0,C 180,E1 17888.848,E2 17888.848} C_VEL
LIN {X 0,Y 517.117,Z 1230.702,A -85,B 0,C 180,E1 17886.404,E2 17886.404} C_VEL
LIN {X 0,Y 519.82,Z 1215.878,A -85,B 0,C 180,E1 17883.371,E2 17883.371} C_VEL
LIN {X 0,Y 522.446,Z 1202.554,A -85,B 0,C 180,E1 17881.002,E2 17881.002} C_VEL
LIN {X 0,Y 525.214,Z 1189.501,A -85,B 0,C 180,E1 17878.939,E2 17878.939} C_VEL
LIN {X 0,Y 528.254,Z 1175.646,A -85,B 0,C 180,E1 17876.964,E2 17876.964} C_VEL
LIN {X 0,Y 532.349,Z 1157.54,A -85,B 0,C 180,E1 17874.653,E2 17874.653} C_VEL
LIN {X 0,Y 536.883,Z 1137.341,A -85,B 0,C 180,E1 17872.413,E2 17872.413} C_VEL
LIN {X 0,Y 540.798,Z 1119.98,A -85,B 0,C 180,E1 17870.708,E2 17870.708} C_VEL
LIN {X 0,Y 544.789,Z 1101.994,A -85,B 0,C 180,E1 17869.128,E2 17869.128} C_VEL
LIN {X 0,Y 549.427,Z 1080.555,A -85,B 0,C 180,E1 17867.46,E2 17867.46} C_VEL
LIN {X 0,Y 554.247,Z 1056.638,A -85,B 0,C 180,E1 17865.863,E2 17865.863} C_VEL
LIN {X 0,Y 557.931,Z 1036.941,A -85,B 0,C 180,E1 17864.716,E2 17864.716} C_VEL
LIN {X 0,Y 561.431,Z 1016.773,A -85,B 0,C 180,E1 17863.69,E2 17863.69} C_VEL
LIN {X 0,Y 564.515,Z 997.425,A -85,B 0,C 180,E1 17862.836,E2 17862.836} C_VEL
LIN {X 0,Y 567.565,Z 976.037,A -85,B 0,C 180,E1 17862.025,E2 17862.025} C_VEL
LIN {X 0,Y 570.859,Z 949.429,A -85,B 0,C 180,E1 17861.198,E2 17861.198} C_VEL
LIN {X 0,Y 573.306,Z 923.608,A -85,B 0,C 180,E1 17860.587,E2 17860.587} C_VEL
LIN {X 0,Y 574.906,Z 901.254,A -85,B 0,C 180,E1 17860.184,E2 17860.184} C_VEL
LIN {X 0,Y 583.208,Z 689.789,A -85,B 0,C 180,E1 17857.064,E2 17857.064} C_VEL
LIN {X 0,Y 589.861,Z 526.411,A -85,B 0,C 180,E1 17854.622,E2 17854.622} C_VEL
LIN {X 0,Y 576.05,Z 505.456,A -85,B 0,C 180,E1 17852.109,E2 17852.109} C_VEL
LIN {X 0,Y 563.527,Z 487.783,A -85,B 0,C 180,E1 17849.585,E2 17849.585} C_VEL
LIN {X 0,Y 553.391,Z 474.306,A -85,B 0,C 180,E1 17847.319,E2 17847.319} C_VEL
LIN {X 0,Y 547.858,Z 467.314,A -85,B 0,C 180,E1 17845.978,E2 17845.978} C_VEL
LIN {X 0,Y 541.135,Z 458.861,A -85,B 0,C 180,E1 17844.218,E2 17844.218} C_VEL
LIN {X 0,Y 537.643,Z 454.891,A -85,B 0,C 180,E1 17843.25,E2 17843.25} C_VEL
LIN {X 0,Y 536.363,Z 453.161,A -85,B 0,C 180,E1 17842.873,E2 17842.873} C_VEL
LIN {X 0,Y 532.998,Z 449.966,A -85,B 0,C 180,E1 17841.892,E2 17841.892} C_VEL
LIN {X 0,Y 531.21,Z 447.016,A -85,B 0,C 180,E1 17841.302,E2 17841.302} C_VEL
LIN {X 0,Y 527.938,Z 444.454,A -85,B 0,C 180,E1 17840.279,E2 17840.279} C_VEL
LIN {X 0,Y 525.79,Z 440.86,A -85,B 0,C 180,E1 17839.496,E2 17839.496} C_VEL
LIN {X 0,Y 522.047,Z 438.153,A -85,B 0,C 180,E1 17838.192,E2 17838.192} C_VEL
LIN {X 0,Y 520.19,Z 434.977,A -85,B 0,C 180,E1 17837.42,E2 17837.42} C_VEL
LIN {X 0,Y 519.78,Z 434,A -85,B 0,C 180,E1 17837.232,E2 17837.232} C_VEL
LIN {X 0,Y 516.413,Z 432.157,A -85,B 0,C 180,E1 17835.901,E2 17835.901} C_VEL
LIN {X 0,Y 514.339,Z 429.343,A -85,B 0,C 180,E1 17834.927,E2 17834.927} C_VEL
LIN {X 0,Y 513.747,Z 427.169,A -85,B 0,C 180,E1 17834.541,E2 17834.541} C_VEL
LIN {X 0,Y 513.775,Z 427.204,A -85,B 0,C 180,E1 17831.109,E2 17831.109} C_VEL
LIN {X 0,Y 513.804,Z 427.176,A -85,B 0,C 180,E1 17827.717,E2 17827.717} C_VEL
LIN {X 0,Y 513.763,Z 427.179,A -85,B 0,C 180,E1 17824.353,E2 17824.353} C_VEL
LIN {X 0,Y 513.792,Z 427.203,A -85,B 0,C 180,E1 17820.892,E2 17820.892} C_VEL
LIN {X 0,Y 513.799,Z 427.16,A -85,B 0,C 180,E1 17817.435,E2 17817.435} C_VEL
LIN {X 0,Y 513.785,Z 427.233,A -85,B 0,C 180,E1 17813.968,E2 17813.968} C_VEL
LIN {X 0,Y 513.788,Z 427.162,A -85,B 0,C 180,E1 17810.478,E2 17810.478} C_VEL
LIN {X 0,Y 513.799,Z 427.202,A -85,B 0,C 180,E1 17807.068,E2 17807.068} C_VEL
LIN {X 0,Y 513.816,Z 427.318,A -85,B 0,C 180,E1 17805.202,E2 17805.202} C_VEL
LIN {X 0,Y 514.614,Z 429.824,A -85,B 0,C 180,E1 17804.735,E2 17804.735} C_VEL
LIN {X 0,Y 516.86,Z 432.541,A -85,B 0,C 180,E1 17803.709,E2 17803.709} C_VEL
LIN {X 0,Y 519.913,Z 434.212,A -85,B 0,C 180,E1 17802.512,E2 17802.512} C_VEL
LIN {X 0,Y 521.448,Z 437.354,A -85,B 0,C 180,E1 17801.844,E2 17801.844} C_VEL
LIN {X 0,Y 524.177,Z 439.875,A -85,B 0,C 180,E1 17800.847,E2 17800.847} C_VEL
LIN {X 0,Y 525.805,Z 440.823,A -85,B 0,C 180,E1 17800.302,E2 17800.302} C_VEL
LIN {X 0,Y 528.032,Z 444.496,A -85,B 0,C 180,E1 17799.493,E2 17799.493} C_VEL
LIN {X 0,Y 531.538,Z 447.452,A -85,B 0,C 180,E1 17798.393,E2 17798.393} C_VEL
LIN {X 0,Y 534.18,Z 451.304,A -85,B 0,C 180,E1 17797.551,E2 17797.551} C_VEL
LIN {X 0,Y 537.079,Z 453.883,A -85,B 0,C 180,E1 17796.725,E2 17796.725} C_VEL
LIN {X 0,Y 540.315,Z 458.086,A -85,B 0,C 180,E1 17795.801,E2 17795.801} C_VEL
LIN {X 0,Y 542.45,Z 460.224,A -85,B 0,C 180,E1 17795.236,E2 17795.236} C_VEL
LIN {X 0,Y 546.1,Z 464.652,A -85,B 0,C 180,E1 17794.282,E2 17794.282} C_VEL
LIN {X 0,Y 547.925,Z 466.875,A -85,B 0,C 180,E1 17793.822,E2 17793.822} C_VEL
LIN {X 0,Y 552.78,Z 472.728,A -85,B 0,C 180,E1 17792.649,E2 17792.649} C_VEL
LIN {X 0,Y 557.721,Z 478.802,A -85,B 0,C 180,E1 17791.517,E2 17791.517} C_VEL
LIN {X 0,Y 565.466,Z 488.51,A -85,B 0,C 180,E1 17789.855,E2 17789.855} C_VEL
LIN {X 0,Y 574.028,Z 499.861,A -85,B 0,C 180,E1 17788.143,E2 17788.143} C_VEL
LIN {X 0,Y 587.632,Z 519.895,A -85,B 0,C 180,E1 17785.633,E2 17785.633} C_VEL
LIN {X 0,Y 589.867,Z 523.675,A -85,B 0,C 180,E1 17785.236,E2 17785.236} C_VEL
LIN {X 0,Y 581.156,Z 737.149,A -85,B 0,C 180,E1 17782.06,E2 17782.06} C_VEL
LIN {X 0,Y 574.911,Z 894.943,A -85,B 0,C 180,E1 17779.73,E2 17779.73} C_VEL
LIN {X 0,Y 573.084,Z 919.854,A -85,B 0,C 180,E1 17779.263,E2 17779.263} C_VEL
LIN {X 0,Y 570.217,Z 947.743,A -85,B 0,C 180,E1 17778.55,E2 17778.55} C_VEL
LIN {X 0,Y 567.483,Z 969.499,A -85,B 0,C 180,E1 17777.848,E2 17777.848} C_VEL
LIN {X 0,Y 564.622,Z 989.53,A -85,B 0,C 180,E1 17777.078,E2 17777.078} C_VEL
LIN {X 0,Y 563.145,Z 999.439,A -85,B 0,C 180,E1 17776.66,E2 17776.66} C_VEL
LIN {X 0,Y 561.28,Z 1006.626,A -85,B 0,C 180,E1 17776.407,E2 17776.407} C_VEL
LIN {X 0,Y 553.792,Z 1024.759,A -85,B 0,C 180,E1 17775.945,E2 17775.945} C_VEL
LIN {X 0,Y 551.814,Z 1031.615,A -85,B 0,C 180,E1 17775.647,E2 17775.647} C_VEL
LIN {X 0,Y 546.551,Z 1057.716,A -85,B 0,C 180,E1 17774.044,E2 17774.044} C_VEL
LIN {X 0,Y 542.224,Z 1077.568,A -85,B 0,C 180,E1 17772.627,E2 17772.627} C_VEL
LIN {X 0,Y 538.192,Z 1095.313,A -85,B 0,C 180,E1 17771.198,E2 17771.198} C_VEL
LIN {X 0,Y 533.914,Z 1113.547,A -85,B 0,C 180,E1 17769.551,E2 17769.551} C_VEL
LIN {X 0,Y 528.614,Z 1135.777,A -85,B 0,C 180,E1 17767.251,E2 17767.251} C_VEL
LIN {X 0,Y 524.443,Z 1152.884,A -85,B 0,C 180,E1 17765.223,E2 17765.223} C_VEL
LIN {X 0,Y 520.966,Z 1167.44,A -85,B 0,C 180,E1 17763.295,E2 17763.295} C_VEL
LIN {X 0,Y 517.554,Z 1182.011,A -85,B 0,C 180,E1 17761.145,E2 17761.145} C_VEL
LIN {X 0,Y 513.856,Z 1198.721,A -85,B 0,C 180,E1 17758.348,E2 17758.348} C_VEL
LIN {X 0,Y 511.043,Z 1212.19,A -85,B 0,C 180,E1 17755.747,E2 17755.747} C_VEL
LIN {X 0,Y 509.114,Z 1222.638,A -85,B 0,C 180,E1 17753.482,E2 17753.482} C_VEL
LIN {X 0,Y 507.521,Z 1232.253,A -85,B 0,C 180,E1 17751.136,E2 17751.136} C_VEL
LIN {X 0,Y 506.072,Z 1242.367,A -85,B 0,C 180,E1 17748.312,E2 17748.312} C_VEL
LIN {X 0,Y 504.993,Z 1251.707,A -85,B 0,C 180,E1 17745.153,E2 17745.153} C_VEL
LIN {X 0,Y 504.455,Z 1257.693,A -85,B 0,C 180,E1 17742.713,E2 17742.713} C_VEL
LIN {X 0,Y 504.156,Z 1262.604,A -85,B 0,C 180,E1 17740.285,E2 17740.285} C_VEL
LIN {X 0,Y 503.968,Z 1266.606,A -85,B 0,C 180,E1 17737.757,E2 17737.757} C_VEL
LIN {X 0,Y 503.926,Z 1269.489,A -85,B 0,C 180,E1 17735.24,E2 17735.24} C_VEL
LIN {X 0,Y 503.909,Z 1271.566,A -85,B 0,C 180,E1 17732.164,E2 17732.164} C_VEL
LIN {X 0,Y 503.866,Z 1271.881,A -85,B 0,C 180,E1 17729.321,E2 17729.321} C_VEL
LIN {X 0,Y 503.91,Z 1271.043,A -85,B 0,C 180,E1 17726.818,E2 17726.818} C_VEL
LIN {X 0,Y 503.93,Z 1269.245,A -85,B 0,C 180,E1 17724.424,E2 17724.424} C_VEL
LIN {X 0,Y 503.98,Z 1266.422,A -85,B 0,C 180,E1 17722.021,E2 17722.021} C_VEL
LIN {X 0,Y 504.174,Z 1262.363,A -85,B 0,C 180,E1 17719.491,E2 17719.491} C_VEL
LIN {X 0,Y 504.576,Z 1256.501,A -85,B 0,C 180,E1 17716.654,E2 17716.654} C_VEL
LIN {X 0,Y 505.37,Z 1248.062,A -85,B 0,C 180,E1 17713.451,E2 17713.451} C_VEL
LIN {X 0,Y 506.32,Z 1240.267,A -85,B 0,C 180,E1 17710.988,E2 17710.988} C_VEL
LIN {X 0,Y 507.599,Z 1231.7,A -85,B 0,C 180,E1 17708.633,E2 17708.633} C_VEL
LIN {X 0,Y 509.308,Z 1221.585,A -85,B 0,C 180,E1 17706.188,E2 17706.188} C_VEL
LIN {X 0,Y 511.931,Z 1208.035,A -85,B 0,C 180,E1 17703.311,E2 17703.311} C_VEL
LIN {X 0,Y 515.032,Z 1193.125,A -85,B 0,C 180,E1 17700.587,E2 17700.587} C_VEL
LIN {X 0,Y 518.005,Z 1180.058,A -85,B 0,C 180,E1 17698.465,E2 17698.465} C_VEL
LIN {X 0,Y 521.221,Z 1166.382,A -85,B 0,C 180,E1 17696.468,E2 17696.468} C_VEL
LIN {X 0,Y 525.165,Z 1149.969,A -85,B 0,C 180,E1 17694.319,E2 17694.319} C_VEL
LIN {X 0,Y 530.189,Z 1129.1,A -85,B 0,C 180,E1 17691.931,E2 17691.931} C_VEL
LIN {X 0,Y 534.428,Z 1111.376,A -85,B 0,C 180,E1 17690.155,E2 17690.155} C_VEL
LIN {X 0,Y 538.49,Z 1094.054,A -85,B 0,C 180,E1 17688.605,E2 17688.605} C_VEL
LIN {X 0,Y 542.921,Z 1074.534,A -85,B 0,C 180,E1 17687.052,E2 17687.052} C_VEL
LIN {X 0,Y 548.451,Z 1048.682,A -85,B 0,C 180,E1 17685.281,E2 17685.281} C_VEL
LIN {X 0,Y 552.459,Z 1028.164,A -85,B 0,C 180,E1 17684.074,E2 17684.074} C_VEL
LIN {X 0,Y 556.087,Z 1008.065,A -85,B 0,C 180,E1 17683.044,E2 17683.044} C_VEL
LIN {X 0,Y 559.476,Z 987.482,A -85,B 0,C 180,E1 17682.132,E2 17682.132} C_VEL
LIN {X 0,Y 563.103,Z 962.722,A -85,B 0,C 180,E1 17681.207,E2 17681.207} C_VEL
LIN {X 0,Y 566.267,Z 935.984,A -85,B 0,C 180,E1 17680.419,E2 17680.419} C_VEL
LIN {X 0,Y 568.377,Z 913.899,A -85,B 0,C 180,E1 17679.907,E2 17679.907} C_VEL
LIN {X 0,Y 569.954,Z 891.906,A -85,B 0,C 180,E1 17679.512,E2 17679.512} C_VEL
LIN {X 0,Y 578.825,Z 675.818,A -85,B 0,C 180,E1 17676.305,E2 17676.305} C_VEL
LIN {X 0,Y 585.143,Z 527.549,A -85,B 0,C 180,E1 17674.075,E2 17674.075} C_VEL
LIN {X 0,Y 573.169,Z 509.688,A -85,B 0,C 180,E1 17671.845,E2 17671.845} C_VEL
LIN {X 0,Y 565.326,Z 498.787,A -85,B 0,C 180,E1 17670.27,E2 17670.27} C_VEL
LIN {X 0,Y 556.509,Z 487.521,A -85,B 0,C 180,E1 17668.375,E2 17668.375} C_VEL
LIN {X 0,Y 552.293,Z 482.275,A -85,B 0,C 180,E1 17667.407,E2 17667.407} C_VEL
LIN {X 0,Y 548.117,Z 477.096,A -85,B 0,C 180,E1 17666.401,E2 17666.401} C_VEL
LIN {X 0,Y 543.992,Z 472.047,A -85,B 0,C 180,E1 17665.358,E2 17665.358} C_VEL
LIN {X 0,Y 540.125,Z 467.249,A -85,B 0,C 180,E1 17664.324,E2 17664.324} C_VEL
LIN {X 0,Y 535.749,Z 462.445,A -85,B 0,C 180,E1 17663.104,E2 17663.104} C_VEL
LIN {X 0,Y 534.312,Z 460.566,A -85,B 0,C 180,E1 17662.675,E2 17662.675} C_VEL
LIN {X 0,Y 530.776,Z 456.938,A -85,B 0,C 180,E1 17661.61,E2 17661.61} C_VEL
LIN {X 0,Y 529.068,Z 454.425,A -85,B 0,C 180,E1 17661.044,E2 17661.044} C_VEL
LIN {X 0,Y 525.745,Z 451.429,A -85,B 0,C 180,E1 17659.961,E2 17659.961} C_VEL
LIN {X 0,Y 523.62,Z 448.14,A -85,B 0,C 180,E1 17659.175,E2 17659.175} C_VEL
LIN {X 0,Y 520.31,Z 445.608,A -85,B 0,C 180,E1 17657.983,E2 17657.983} C_VEL
LIN {X 0,Y 518.275,Z 442.06,A -85,B 0,C 180,E1 17657.11,E2 17657.11} C_VEL
LIN {X 0,Y 514.404,Z 439.283,A -85,B 0,C 180,E1 17655.502,E2 17655.502} C_VEL
LIN {X 0,Y 512.501,Z 436.267,A -85,B 0,C 180,E1 17654.548,E2 17654.548} C_VEL
LIN {X 0,Y 511.974,Z 434.972,A -85,B 0,C 180,E1 17654.246,E2 17654.246} C_VEL
LIN {X 0,Y 508.3,Z 433.086,A -85,B 0,C 180,E1 17652.381,E2 17652.381} C_VEL
LIN {X 0,Y 506.25,Z 429.97,A -85,B 0,C 180,E1 17651.045,E2 17651.045} C_VEL
LIN {X 0,Y 505.795,Z 428.182,A -85,B 0,C 180,E1 17650.594,E2 17650.594} C_VEL
LIN {X 0,Y 505.841,Z 428.176,A -85,B 0,C 180,E1 17647.154,E2 17647.154} C_VEL
LIN {X 0,Y 505.802,Z 428.161,A -85,B 0,C 180,E1 17643.854,E2 17643.854} C_VEL
LIN {X 0,Y 505.796,Z 428.21,A -85,B 0,C 180,E1 17640.34,E2 17640.34} C_VEL
LIN {X 0,Y 505.845,Z 428.147,A -85,B 0,C 180,E1 17637.054,E2 17637.054} C_VEL
LIN {X 0,Y 505.798,Z 428.229,A -85,B 0,C 180,E1 17633.644,E2 17633.644} C_VEL
LIN {X 0,Y 505.791,Z 428.156,A -85,B 0,C 180,E1 17630.096,E2 17630.096} C_VEL
LIN {X 0,Y 505.825,Z 428.416,A -85,B 0,C 180,E1 17629.431,E2 17629.431} C_VEL
LIN {X 0,Y 506.786,Z 431.07,A -85,B 0,C 180,E1 17628.678,E2 17628.678} C_VEL
LIN {X 0,Y 508.877,Z 433.588,A -85,B 0,C 180,E1 17627.402,E2 17627.402} C_VEL
LIN {X 0,Y 512.166,Z 435.312,A -85,B 0,C 180,E1 17625.76,E2 17625.76} C_VEL
LIN {X 0,Y 513.7,Z 438.425,A -85,B 0,C 180,E1 17624.939,E2 17624.939} C_VEL
LIN {X 0,Y 516.51,Z 441.04,A -85,B 0,C 180,E1 17623.698,E2 17623.698} C_VEL
LIN {X 0,Y 518.254,Z 442.089,A -85,B 0,C 180,E1 17623.004,E2 17623.004} C_VEL
LIN {X 0,Y 520.248,Z 445.577,A -85,B 0,C 180,E1 17622.148,E2 17622.148} C_VEL
LIN {X 0,Y 523.292,Z 447.99,A -85,B 0,C 180,E1 17621.045,E2 17621.045} C_VEL
LIN {X 0,Y 524.103,Z 448.771,A -85,B 0,C 180,E1 17620.757,E2 17620.757} C_VEL
LIN {X 0,Y 526.632,Z 452.482,A -85,B 0,C 180,E1 17619.842,E2 17619.842} C_VEL
LIN {X 0,Y 529.605,Z 455.042,A -85,B 0,C 180,E1 17618.891,E2 17618.891} C_VEL
LIN {X 0,Y 532.553,Z 459.093,A -85,B 0,C 180,E1 17617.944,E2 17617.944} C_VEL
LIN {X 0,Y 535.062,Z 461.413,A -85,B 0,C 180,E1 17617.214,E2 17617.214} C_VEL
LIN {X 0,Y 538.624,Z 465.856,A -85,B 0,C 180,E1 17616.186,E2 17616.186} C_VEL
LIN {X 0,Y 540.89,Z 468.474,A -85,B 0,C 180,E1 17615.567,E2 17615.567} C_VEL
LIN {X 0,Y 547.932,Z 477.504,A -85,B 0,C 180,E1 17613.735,E2 17613.735} C_VEL
LIN {X 0,Y 555.845,Z 487.892,A -85,B 0,C 180,E1 17611.852,E2 17611.852} C_VEL
LIN {X 0,Y 566.186,Z 502.254,A -85,B 0,C 180,E1 17609.605,E2 17609.605} C_VEL
LIN {X 0,Y 576.368,Z 517.155,A -85,B 0,C 180,E1 17607.584,E2 17607.584} C_VEL
LIN {X 0,Y 585.215,Z 530.994,A -85,B 0,C 180,E1 17605.95,E2 17605.95} C_VEL
LIN {X 0,Y 576.006,Z 748.398,A -85,B 0,C 180,E1 17602.701,E2 17602.701} C_VEL
LIN {X 0,Y 569.662,Z 903.026,A -85,B 0,C 180,E1 17600.405,E2 17600.405} C_VEL
LIN {X 0,Y 567.694,Z 928.68,A -85,B 0,C 180,E1 17599.925,E2 17599.925} C_VEL
LIN {X 0,Y 564.702,Z 956.343,A -85,B 0,C 180,E1 17599.216,E2 17599.216} C_VEL
LIN {X 0,Y 561.868,Z 978.097,A -85,B 0,C 180,E1 17598.514,E2 17598.514} C_VEL
LIN {X 0,Y 558.781,Z 998.842,A -85,B 0,C 180,E1 17597.715,E2 17597.715} C_VEL
LIN {X 0,Y 555.407,Z 1019.095,A -85,B 0,C 180,E1 17596.805,E2 17596.805} C_VEL
LIN {X 0,Y 550.886,Z 1044.009,A -85,B 0,C 180,E1 17595.498,E2 17595.498} C_VEL
LIN {X 0,Y 546.031,Z 1067.725,A -85,B 0,C 180,E1 17594.015,E2 17594.015} C_VEL
LIN {X 0,Y 541.982,Z 1086.458,A -85,B 0,C 180,E1 17592.68,E2 17592.68} C_VEL
LIN {X 0,Y 537.878,Z 1104.696,A -85,B 0,C 180,E1 17591.217,E2 17591.217} C_VEL
LIN {X 0,Y 533.292,Z 1124.551,A -85,B 0,C 180,E1 17589.423,E2 17589.423} C_VEL
LIN {X 0,Y 528.123,Z 1146.39,A -85,B 0,C 180,E1 17587.148,E2 17587.148} C_VEL
LIN {X 0,Y 524.244,Z 1162.618,A -85,B 0,C 180,E1 17585.231,E2 17585.231} C_VEL
LIN {X 0,Y 520.806,Z 1177.302,A -85,B 0,C 180,E1 17583.299,E2 17583.299} C_VEL
LIN {X 0,Y 517.482,Z 1191.778,A -85,B 0,C 180,E1 17581.182,E2 17581.182} C_VEL
LIN {X 0,Y 513.864,Z 1208.491,A -85,B 0,C 180,E1 17578.416,E2 17578.416} C_VEL
LIN {X 0,Y 511.229,Z 1221.278,A -85,B 0,C 180,E1 17575.978,E2 17575.978} C_VEL
LIN {X 0,Y 509.179,Z 1232.267,A -85,B 0,C 180,E1 17573.611,E2 17573.611} C_VEL
LIN {X 0,Y 507.558,Z 1241.988,A -85,B 0,C 180,E1 17571.248,E2 17571.248} C_VEL
LIN {X 0,Y 506.196,Z 1251.33,A -85,B 0,C 180,E1 17568.658,E2 17568.658} C_VEL
LIN {X 0,Y 505.05,Z 1261.237,A -85,B 0,C 180,E1 17565.38,E2 17565.38} C_VEL
LIN {X 0,Y 504.464,Z 1267.624,A -85,B 0,C 180,E1 17562.789,E2 17562.789} C_VEL
LIN {X 0,Y 504.161,Z 1272.557,A -85,B 0,C 180,E1 17560.356,E2 17560.356} C_VEL
LIN {X 0,Y 503.973,Z 1276.519,A -85,B 0,C 180,E1 17557.865,E2 17557.865} C_VEL
LIN {X 0,Y 503.93,Z 1279.314,A -85,B 0,C 180,E1 17555.462,E2 17555.462} C_VEL
LIN {X 0,Y 503.909,Z 1281.22,A -85,B 0,C 180,E1 17552.84,E2 17552.84} C_VEL
LIN {X 0,Y 503.883,Z 1281.961,A -85,B 0,C 180,E1 17549.769,E2 17549.769} C_VEL
LIN {X 0,Y 503.911,Z 1281.148,A -85,B 0,C 180,E1 17547.04,E2 17547.04} C_VEL
LIN {X 0,Y 503.928,Z 1279.306,A -85,B 0,C 180,E1 17544.532,E2 17544.532} C_VEL
LIN {X 0,Y 503.974,Z 1276.509,A -85,B 0,C 180,E1 17542.129,E2 17542.129} C_VEL
LIN {X 0,Y 504.167,Z 1272.477,A -85,B 0,C 180,E1 17539.6,E2 17539.6} C_VEL
LIN {X 0,Y 504.496,Z 1267.283,A -85,B 0,C 180,E1 17537.055,E2 17537.055} C_VEL
LIN {X 0,Y 505.239,Z 1259.317,A -85,B 0,C 180,E1 17533.912,E2 17533.912} C_VEL
LIN {X 0,Y 506.299,Z 1250.436,A -85,B 0,C 180,E1 17531.082,E2 17531.082} C_VEL
LIN {X 0,Y 507.582,Z 1241.839,A -85,B 0,C 180,E1 17528.713,E2 17528.713} C_VEL
LIN {X 0,Y 509.188,Z 1232.244,A -85,B 0,C 180,E1 17526.382,E2 17526.382} C_VEL
LIN {X 0,Y 511.358,Z 1220.678,A -85,B 0,C 180,E1 17523.897,E2 17523.897} C_VEL
LIN {X 0,Y 514.613,Z 1204.773,A -85,B 0,C 180,E1 17520.936,E2 17520.936} C_VEL
LIN {X 0,Y 517.82,Z 1190.295,A -85,B 0,C 180,E1 17518.593,E2 17518.593} C_VEL
LIN {X 0,Y 521.016,Z 1176.403,A -85,B 0,C 180,E1 17516.577,E2 17516.577} C_VEL
LIN {X 0,Y 524.591,Z 1161.17,A -85,B 0,C 180,E1 17514.587,E2 17514.587} C_VEL
LIN {X 0,Y 529.379,Z 1141.152,A -85,B 0,C 180,E1 17512.266,E2 17512.266} C_VEL
LIN {X 0,Y 534.055,Z 1121.188,A -85,B 0,C 180,E1 17510.262,E2 17510.262} C_VEL
LIN {X 0,Y 538.203,Z 1103.269,A -85,B 0,C 180,E1 17508.663,E2 17508.663} C_VEL
LIN {X 0,Y 542.494,Z 1084.148,A -85,B 0,C 180,E1 17507.146,E2 17507.146} C_VEL
LIN {X 0,Y 547.654,Z 1060.155,A -85,B 0,C 180,E1 17505.484,E2 17505.484} C_VEL
LIN {X 0,Y 552.001,Z 1037.855,A -85,B 0,C 180,E1 17504.166,E2 17504.166} C_VEL
LIN {X 0,Y 555.687,Z 1017.419,A -85,B 0,C 180,E1 17503.116,E2 17503.116} C_VEL
LIN {X 0,Y 559.007,Z 997.33,A -85,B 0,C 180,E1 17502.223,E2 17502.223} C_VEL
LIN {X 0,Y 562.192,Z 975.769,A -85,B 0,C 180,E1 17501.405,E2 17501.405} C_VEL
LIN {X 0,Y 565.586,Z 949.214,A -85,B 0,C 180,E1 17500.58,E2 17500.58} C_VEL
LIN {X 0,Y 568.102,Z 923.537,A -85,B 0,C 180,E1 17499.972,E2 17499.972} C_VEL
LIN {X 0,Y 569.749,Z 901.19,A -85,B 0,C 180,E1 17499.567,E2 17499.567} C_VEL
LIN {X 0,Y 578.367,Z 690.317,A -85,B 0,C 180,E1 17496.438,E2 17496.438} C_VEL
LIN {X 0,Y 585.095,Z 530.675,A -85,B 0,C 180,E1 17494.034,E2 17494.034} C_VEL
LIN {X 0,Y 572.763,Z 511.688,A -85,B 0,C 180,E1 17491.729,E2 17491.729} C_VEL
LIN {X 0,Y 560.392,Z 494.084,A -85,B 0,C 180,E1 17489.18,E2 17489.18} C_VEL
LIN {X 0,Y 550.703,Z 481.106,A -85,B 0,C 180,E1 17486.966,E2 17486.966} C_VEL
LIN {X 0,Y 545.347,Z 474.224,A -85,B 0,C 180,E1 17485.639,E2 17485.639} C_VEL
LIN {X 0,Y 538.892,Z 466.09,A -85,B 0,C 180,E1 17483.917,E2 17483.917} C_VEL
LIN {X 0,Y 535.292,Z 461.771,A -85,B 0,C 180,E1 17482.892,E2 17482.892} C_VEL
LIN {X 0,Y 533.999,Z 460.351,A -85,B 0,C 180,E1 17482.515,E2 17482.515} C_VEL
LIN {X 0,Y 530.566,Z 456.651,A -85,B 0,C 180,E1 17481.474,E2 17481.474} C_VEL
LIN {X 0,Y 529.26,Z 454.542,A -85,B 0,C 180,E1 17481.036,E2 17481.036} C_VEL
LIN {X 0,Y 525.901,Z 451.633,A -85,B 0,C 180,E1 17479.955,E2 17479.955} C_VEL
LIN {X 0,Y 523.774,Z 448.214,A -85,B 0,C 180,E1 17479.169,E2 17479.169} C_VEL
LIN {X 0,Y 520.524,Z 445.851,A -85,B 0,C 180,E1 17478.015,E2 17478.015} C_VEL
LIN {X 0,Y 518.363,Z 442.288,A -85,B 0,C 180,E1 17477.107,E2 17477.107} C_VEL
LIN {X 0,Y 517.989,Z 441.712,A -85,B 0,C 180,E1 17476.947,E2 17476.947} C_VEL
LIN {X 0,Y 514.713,Z 439.606,A -85,B 0,C 180,E1 17475.608,E2 17475.608} C_VEL
LIN {X 0,Y 512.644,Z 436.599,A -85,B 0,C 180,E1 17474.602,E2 17474.602} C_VEL
LIN {X 0,Y 512.022,Z 434.977,A -85,B 0,C 180,E1 17474.244,E2 17474.244} C_VEL
LIN {X 0,Y 508.306,Z 433.074,A -85,B 0,C 180,E1 17472.381,E2 17472.381} C_VEL
LIN {X 0,Y 506.307,Z 430.074,A -85,B 0,C 180,E1 17471.102,E2 17471.102} C_VEL
LIN {X 0,Y 505.818,Z 428.176,A -85,B 0,C 180,E1 17470.651,E2 17470.651} C_VEL
LIN {X 0,Y 505.853,Z 428.181,A -85,B 0,C 180,E1 17467.154,E2 17467.154} C_VEL
LIN {X 0,Y 505.853,Z 428.15,A -85,B 0,C 180,E1 17463.74,E2 17463.74} C_VEL
LIN {X 0,Y 505.837,Z 428.221,A -85,B 0,C 180,E1 17460.227,E2 17460.227} C_VEL
LIN {X 0,Y 505.848,Z 428.146,A -85,B 0,C 180,E1 17456.714,E2 17456.714} C_VEL
LIN {X 0,Y 505.866,Z 428.196,A -85,B 0,C 180,E1 17453.189,E2 17453.189} C_VEL
LIN {X 0,Y 505.852,Z 428.161,A -85,B 0,C 180,E1 17449.637,E2 17449.637} C_VEL
LIN {X 0,Y 505.892,Z 428.403,A -85,B 0,C 180,E1 17449.062,E2 17449.062} C_VEL
LIN {X 0,Y 506.824,Z 431.148,A -85,B 0,C 180,E1 17448.333,E2 17448.333} C_VEL
LIN {X 0,Y 509.17,Z 433.722,A -85,B 0,C 180,E1 17446.948,E2 17446.948} C_VEL
LIN {X 0,Y 512.19,Z 435.188,A -85,B 0,C 180,E1 17445.472,E2 17445.472} C_VEL
LIN {X 0,Y 513.612,Z 438.28,A -85,B 0,C 180,E1 17444.705,E2 17444.705} C_VEL
LIN {X 0,Y 516.431,Z 440.955,A -85,B 0,C 180,E1 17443.464,E2 17443.464} C_VEL
LIN {X 0,Y 518.244,Z 442.025,A -85,B 0,C 180,E1 17442.748,E2 17442.748} C_VEL
LIN {X 0,Y 520.333,Z 445.579,A -85,B 0,C 180,E1 17441.862,E2 17441.862} C_VEL
LIN {X 0,Y 523.552,Z 448.089,A -85,B 0,C 180,E1 17440.707,E2 17440.707} C_VEL
LIN {X 0,Y 524.343,Z 449.126,A -85,B 0,C 180,E1 17440.419,E2 17440.419} C_VEL
LIN {X 0,Y 527.07,Z 452.86,A -85,B 0,C 180,E1 17439.454,E2 17439.454} C_VEL
LIN {X 0,Y 529.667,Z 455.047,A -85,B 0,C 180,E1 17438.633,E2 17438.633} C_VEL
LIN {X 0,Y 532.715,Z 459.195,A -85,B 0,C 180,E1 17437.661,E2 17437.661} C_VEL
LIN {X 0,Y 535.147,Z 461.459,A -85,B 0,C 180,E1 17436.956,E2 17436.956} C_VEL
LIN {X 0,Y 538.636,Z 465.804,A -85,B 0,C 180,E1 17435.954,E2 17435.954} C_VEL
LIN {X 0,Y 540.375,Z 467.656,A -85,B 0,C 180,E1 17435.484,E2 17435.484} C_VEL
LIN {X 0,Y 544.383,Z 472.374,A -85,B 0,C 180,E1 17434.429,E2 17434.429} C_VEL
LIN {X 0,Y 550.899,Z 480.552,A -85,B 0,C 180,E1 17432.811,E2 17432.811} C_VEL
LIN {X 0,Y 555.394,Z 486.093,A -85,B 0,C 180,E1 17431.768,E2 17431.768} C_VEL
LIN {X 0,Y 563.173,Z 496.002,A -85,B 0,C 180,E1 17430.072,E2 17430.072} C_VEL
LIN {X 0,Y 571.097,Z 506.605,A -85,B 0,C 180,E1 17428.462,E2 17428.462} C_VEL
LIN {X 0,Y 584.441,Z 526.472,A -85,B 0,C 180,E1 17425.953,E2 17425.953} C_VEL
LIN {X 0,Y 585.144,Z 527.952,A -85,B 0,C 180,E1 17425.819,E2 17425.819} C_VEL
LIN {X 0,Y 576.092,Z 741.34,A -85,B 0,C 180,E1 17422.629,E2 17422.629} C_VEL
LIN {X 0,Y 569.76,Z 895.057,A -85,B 0,C 180,E1 17420.345,E2 17420.345} C_VEL
LIN {X 0,Y 567.85,Z 920.242,A -85,B 0,C 180,E1 17419.872,E2 17419.872} C_VEL
LIN {X 0,Y 564.885,Z 948.062,A -85,B 0,C 180,E1 17419.157,E2 17419.157} C_VEL
LIN {X 0,Y 562.052,Z 969.86,A -85,B 0,C 180,E1 17418.45,E2 17418.45} C_VEL
LIN {X 0,Y 559.129,Z 989.63,A -85,B 0,C 180,E1 17417.687,E2 17417.687} C_VEL
LIN {X 0,Y 555.757,Z 1009.948,A -85,B 0,C 180,E1 17416.775,E2 17416.775} C_VEL
LIN {X 0,Y 551.814,Z 1031.615,A -85,B 0,C 180,E1 17415.647,E2 17415.647} C_VEL
LIN {X 0,Y 549.791,Z 1038.501,A -85,B 0,C 180,E1 17415.333,E2 17415.333} C_VEL
LIN {X 0,Y 541.789,Z 1056.023,A -85,B 0,C 180,E1 17414.699,E2 17414.699} C_VEL
LIN {X 0,Y 539.639,Z 1062.49,A -85,B 0,C 180,E1 17414.327,E2 17414.327} C_VEL
LIN {X 0,Y 535.109,Z 1082.399,A -85,B 0,C 180,E1 17412.858,E2 17412.858} C_VEL
LIN {X 0,Y 529.367,Z 1106.377,A -85,B 0,C 180,E1 17410.811,E2 17410.811} C_VEL
LIN {X 0,Y 524.86,Z 1124.424,A -85,B 0,C 180,E1 17409.039,E2 17409.039} C_VEL
LIN {X 0,Y 520.814,Z 1140.412,A -85,B 0,C 180,E1 17407.282,E2 17407.282} C_VEL
LIN {X 0,Y 516.934,Z 1155.743,A -85,B 0,C 180,E1 17405.404,E2 17405.404} C_VEL
LIN {X 0,Y 512.549,Z 1173.419,A -85,B 0,C 180,E1 17402.977,E2 17402.977} C_VEL
LIN {X 0,Y 508.495,Z 1190.119,A -85,B 0,C 180,E1 17400.318,E2 17400.318} C_VEL
LIN {X 0,Y 505.626,Z 1202.601,A -85,B 0,C 180,E1 17398.079,E2 17398.079} C_VEL
LIN {X 0,Y 503.167,Z 1213.96,A -85,B 0,C 180,E1 17395.8,E2 17395.8} C_VEL
LIN {X 0,Y 500.741,Z 1226.688,A -85,B 0,C 180,E1 17392.918,E2 17392.918} C_VEL
LIN {X 0,Y 498.853,Z 1237.916,A -85,B 0,C 180,E1 17389.925,E2 17389.925} C_VEL
LIN {X 0,Y 497.708,Z 1246.085,A -85,B 0,C 180,E1 17387.393,E2 17387.393} C_VEL
LIN {X 0,Y 496.966,Z 1252.641,A -85,B 0,C 180,E1 17385.037,E2 17385.037} C_VEL
LIN {X 0,Y 496.437,Z 1258.457,A -85,B 0,C 180,E1 17382.567,E2 17382.567} C_VEL
LIN {X 0,Y 496.129,Z 1263.221,A -85,B 0,C 180,E1 17380.101,E2 17380.101} C_VEL
LIN {X 0,Y 495.978,Z 1267.563,A -85,B 0,C 180,E1 17377.183,E2 17377.183} C_VEL
LIN {X 0,Y 495.917,Z 1270.508,A -85,B 0,C 180,E1 17374.05,E2 17374.05} C_VEL
LIN {X 0,Y 495.905,Z 1271.703,A -85,B 0,C 180,E1 17371.505,E2 17371.505} C_VEL
LIN {X 0,Y 495.869,Z 1271.835,A -85,B 0,C 180,E1 17369.079,E2 17369.079} C_VEL
LIN {X 0,Y 495.91,Z 1271.042,A -85,B 0,C 180,E1 17366.767,E2 17366.767} C_VEL
LIN {X 0,Y 495.934,Z 1269.242,A -85,B 0,C 180,E1 17364.334,E2 17364.334} C_VEL
LIN {X 0,Y 495.989,Z 1266.418,A -85,B 0,C 180,E1 17361.891,E2 17361.891} C_VEL
LIN {X 0,Y 496.197,Z 1262.359,A -85,B 0,C 180,E1 17359.32,E2 17359.32} C_VEL
LIN {X 0,Y 496.612,Z 1256.631,A -85,B 0,C 180,E1 17356.498,E2 17356.498} C_VEL
LIN {X 0,Y 497.444,Z 1248.412,A -85,B 0,C 180,E1 17353.3,E2 17353.3} C_VEL
LIN {X 0,Y 498.492,Z 1240.263,A -85,B 0,C 180,E1 17350.677,E2 17350.677} C_VEL
LIN {X 0,Y 499.856,Z 1231.695,A -85,B 0,C 180,E1 17348.285,E2 17348.285} C_VEL
LIN {X 0,Y 501.607,Z 1221.936,A -85,B 0,C 180,E1 17345.885,E2 17345.885} C_VEL
LIN {X 0,Y 504.202,Z 1209.266,A -85,B 0,C 180,E1 17343.123,E2 17343.123} C_VEL
LIN {X 0,Y 507.593,Z 1193.909,A -85,B 0,C 180,E1 17340.243,E2 17340.243} C_VEL
LIN {X 0,Y 510.688,Z 1180.911,A -85,B 0,C 180,E1 17338.092,E2 17338.092} C_VEL
LIN {X 0,Y 514.041,Z 1167.309,A -85,B 0,C 180,E1 17336.07,E2 17336.07} C_VEL
LIN {X 0,Y 517.811,Z 1152.26,A -85,B 0,C 180,E1 17334.06,E2 17334.06} C_VEL
LIN {X 0,Y 522.852,Z 1132.5,A -85,B 0,C 180,E1 17331.719,E2 17331.719} C_VEL
LIN {X 0,Y 527.774,Z 1112.671,A -85,B 0,C 180,E1 17329.692,E2 17329.692} C_VEL
LIN {X 0,Y 532.102,Z 1094.962,A -85,B 0,C 180,E1 17328.085,E2 17328.085} C_VEL
LIN {X 0,Y 536.303,Z 1077.162,A -85,B 0,C 180,E1 17326.646,E2 17326.646} C_VEL
LIN {X 0,Y 540.978,Z 1056.477,A -85,B 0,C 180,E1 17325.167,E2 17325.167} C_VEL
LIN {X 0,Y 546.275,Z 1030.985,A -85,B 0,C 180,E1 17323.608,E2 17323.608} C_VEL
LIN {X 0,Y 550.358,Z 1009.272,A -85,B 0,C 180,E1 17322.478,E2 17322.478} C_VEL
LIN {X 0,Y 553.648,Z 990.124,A -85,B 0,C 180,E1 17321.617,E2 17321.617} C_VEL
LIN {X 0,Y 556.819,Z 969.423,A -85,B 0,C 180,E1 17320.817,E2 17320.817} C_VEL
LIN {X 0,Y 559.863,Z 946.612,A -85,B 0,C 180,E1 17320.081,E2 17320.081} C_VEL
LIN {X 0,Y 562.927,Z 917.834,A -85,B 0,C 180,E1 17319.359,E2 17319.359} C_VEL
LIN {X 0,Y 564.736,Z 894.451,A -85,B 0,C 180,E1 17318.924,E2 17318.924} C_VEL
LIN {X 0,Y 573.491,Z 690.077,A -85,B 0,C 180,E1 17315.872,E2 17315.872} C_VEL
LIN {X 0,Y 580.5,Z 531.829,A -85,B 0,C 180,E1 17313.484,E2 17313.484} C_VEL
LIN {X 0,Y 567.566,Z 512.492,A -85,B 0,C 180,E1 17310.988,E2 17310.988} C_VEL
LIN {X 0,Y 561.388,Z 504.151,A -85,B 0,C 180,E1 17309.709,E2 17309.709} C_VEL
LIN {X 0,Y 553.876,Z 494.411,A -85,B 0,C 180,E1 17308.052,E2 17308.052} C_VEL
LIN {X 0,Y 549.31,Z 488.7,A -85,B 0,C 180,E1 17306.982,E2 17306.982} C_VEL
LIN {X 0,Y 545.491,Z 483.924,A -85,B 0,C 180,E1 17306.041,E2 17306.041} C_VEL
LIN {X 0,Y 541.516,Z 479.039,A -85,B 0,C 180,E1 17305.014,E2 17305.014} C_VEL
LIN {X 0,Y 537.16,Z 473.726,A -85,B 0,C 180,E1 17303.824,E2 17303.824} C_VEL
LIN {X 0,Y 533.333,Z 469.207,A -85,B 0,C 180,E1 17302.719,E2 17302.719} C_VEL
LIN {X 0,Y 531.629,Z 467.43,A -85,B 0,C 180,E1 17302.213,E2 17302.213} C_VEL
LIN {X 0,Y 528.223,Z 463.369,A -85,B 0,C 180,E1 17301.137,E2 17301.137} C_VEL
LIN {X 0,Y 527.142,Z 461.914,A -85,B 0,C 180,E1 17300.775,E2 17300.775} C_VEL
LIN {X 0,Y 523.663,Z 458.494,A -85,B 0,C 180,E1 17299.608,E2 17299.608} C_VEL
LIN {X 0,Y 522.071,Z 455.871,A -85,B 0,C 180,E1 17299.001,E2 17299.001} C_VEL
LIN {X 0,Y 518.756,Z 453.26,A -85,B 0,C 180,E1 17297.789,E2 17297.789} C_VEL
LIN {X 0,Y 516.389,Z 449.457,A -85,B 0,C 180,E1 17296.769,E2 17296.769} C_VEL
LIN {X 0,Y 513.081,Z 447.102,A -85,B 0,C 180,E1 17295.369,E2 17295.369} C_VEL
LIN {X 0,Y 510.928,Z 443.761,A -85,B 0,C 180,E1 17294.275,E2 17294.275} C_VEL
LIN {X 0,Y 510.555,Z 442.803,A -85,B 0,C 180,E1 17294.055,E2 17294.055} C_VEL
LIN {X 0,Y 506.952,Z 440.795,A -85,B 0,C 180,E1 17292.184,E2 17292.184} C_VEL
LIN {X 0,Y 504.869,Z 437.517,A -85,B 0,C 180,E1 17290.787,E2 17290.787} C_VEL
LIN {X 0,Y 504.406,Z 436.054,A -85,B 0,C 180,E1 17290.393,E2 17290.393} C_VEL
LIN {X 0,Y 500.503,Z 434.106,A -85,B 0,C 180,E1 17287.346,E2 17287.346} C_VEL
LIN {X 0,Y 498.211,Z 430.732,A -85,B 0,C 180,E1 17284.259,E2 17284.259} C_VEL
LIN {X 0,Y 497.907,Z 429.134,A -85,B 0,C 180,E1 17283.223,E2 17283.223} C_VEL
LIN {X 0,Y 497.859,Z 429.217,A -85,B 0,C 180,E1 17279.885,E2 17279.885} C_VEL
LIN {X 0,Y 497.911,Z 429.366,A -85,B 0,C 180,E1 17276.661,E2 17276.661} C_VEL
LIN {X 0,Y 499.271,Z 432.845,A -85,B 0,C 180,E1 17274.138,E2 17274.138} C_VEL
LIN {X 0,Y 502.915,Z 435.592,A -85,B 0,C 180,E1 17270.733,E2 17270.733} C_VEL
LIN {X 0,Y 504.465,Z 436.226,A -85,B 0,C 180,E1 17269.666,E2 17269.666} C_VEL
LIN {X 0,Y 505.948,Z 439.591,A -85,B 0,C 180,E1 17268.55,E2 17268.55} C_VEL
LIN {X 0,Y 508.538,Z 441.98,A -85,B 0,C 180,E1 17267.047,E2 17267.047} C_VEL
LIN {X 0,Y 510.682,Z 443.142,A -85,B 0,C 180,E1 17265.978,E2 17265.978} C_VEL
LIN {X 0,Y 512.606,Z 446.554,A -85,B 0,C 180,E1 17264.964,E2 17264.964} C_VEL
LIN {X 0,Y 515.564,Z 449.063,A -85,B 0,C 180,E1 17263.667,E2 17263.667} C_VEL
LIN {X 0,Y 516.621,Z 449.798,A -85,B 0,C 180,E1 17263.239,E2 17263.239} C_VEL
LIN {X 0,Y 518.871,Z 453.432,A -85,B 0,C 180,E1 17262.273,E2 17262.273} C_VEL
LIN {X 0,Y 522.325,Z 456.319,A -85,B 0,C 180,E1 17261.008,E2 17261.008} C_VEL
LIN {X 0,Y 525.209,Z 460.336,A -85,B 0,C 180,E1 17259.959,E2 17259.959} C_VEL
LIN {X 0,Y 527.826,Z 462.727,A -85,B 0,C 180,E1 17259.108,E2 17259.108} C_VEL
LIN {X 0,Y 531.094,Z 466.965,A -85,B 0,C 180,E1 17258.055,E2 17258.055} C_VEL
LIN {X 0,Y 533.144,Z 468.961,A -85,B 0,C 180,E1 17257.447,E2 17257.447} C_VEL
LIN {X 0,Y 536.95,Z 473.566,A -85,B 0,C 180,E1 17256.341,E2 17256.341} C_VEL
LIN {X 0,Y 545.13,Z 483.953,A -85,B 0,C 180,E1 17254.145,E2 17254.145} C_VEL
LIN {X 0,Y 553.622,Z 495.374,A -85,B 0,C 180,E1 17252.08,E2 17252.08} C_VEL
LIN {X 0,Y 563.328,Z 508.985,A -85,B 0,C 180,E1 17249.935,E2 17249.935} C_VEL
LIN {X 0,Y 573.397,Z 523.891,A -85,B 0,C 180,E1 17247.898,E2 17247.898} C_VEL
LIN {X 0,Y 580.553,Z 535.272,A -85,B 0,C 180,E1 17246.541,E2 17246.541} C_VEL
LIN {X 0,Y 570.961,Z 753.26,A -85,B 0,C 180,E1 17243.27,E2 17243.27} C_VEL
LIN {X 0,Y 564.573,Z 902.969,A -85,B 0,C 180,E1 17241.033,E2 17241.033} C_VEL
LIN {X 0,Y 562.518,Z 928.929,A -85,B 0,C 180,E1 17240.546,E2 17240.546} C_VEL
LIN {X 0,Y 559.432,Z 956.452,A -85,B 0,C 180,E1 17239.837,E2 17239.837} C_VEL
LIN {X 0,Y 556.529,Z 978.015,A -85,B 0,C 180,E1 17239.139,E2 17239.139} C_VEL
LIN {X 0,Y 553.32,Z 998.845,A -85,B 0,C 180,E1 17238.335,E2 17238.335} C_VEL
LIN {X 0,Y 549.841,Z 1019.011,A -85,B 0,C 180,E1 17237.426,E2 17237.426} C_VEL
LIN {X 0,Y 545.112,Z 1044.123,A -85,B 0,C 180,E1 17236.103,E2 17236.103} C_VEL
LIN {X 0,Y 540.112,Z 1067.638,A -85,B 0,C 180,E1 17234.625,E2 17234.625} C_VEL
LIN {X 0,Y 535.74,Z 1087.107,A -85,B 0,C 180,E1 17233.225,E2 17233.225} C_VEL
LIN {X 0,Y 531.169,Z 1106.617,A -85,B 0,C 180,E1 17231.637,E2 17231.637} C_VEL
LIN {X 0,Y 525.583,Z 1129.697,A -85,B 0,C 180,E1 17229.48,E2 17229.48} C_VEL
LIN {X 0,Y 521.066,Z 1147.825,A -85,B 0,C 180,E1 17227.53,E2 17227.53} C_VEL
LIN {X 0,Y 517.162,Z 1163.456,A -85,B 0,C 180,E1 17225.651,E2 17225.651} C_VEL
LIN {X 0,Y 513.583,Z 1178.06,A -85,B 0,C 180,E1 17223.696,E2 17223.696} C_VEL
LIN {X 0,Y 509.576,Z 1194.855,A -85,B 0,C 180,E1 17221.182,E2 17221.182} C_VEL
LIN {X 0,Y 505.944,Z 1210.768,A -85,B 0,C 180,E1 17218.424,E2 17218.424} C_VEL
LIN {X 0,Y 503.341,Z 1222.947,A -85,B 0,C 180,E1 17216.036,E2 17216.036} C_VEL
LIN {X 0,Y 501.345,Z 1233.295,A -85,B 0,C 180,E1 17213.753,E2 17213.753} C_VEL
LIN {X 0,Y 499.528,Z 1243.822,A -85,B 0,C 180,E1 17211.114,E2 17211.114} C_VEL
LIN {X 0,Y 497.863,Z 1254.926,A -85,B 0,C 180,E1 17207.83,E2 17207.83} C_VEL
LIN {X 0,Y 497.03,Z 1262.145,A -85,B 0,C 180,E1 17205.276,E2 17205.276} C_VEL
LIN {X 0,Y 496.473,Z 1268.06,A -85,B 0,C 180,E1 17202.795,E2 17202.795} C_VEL
LIN {X 0,Y 496.159,Z 1272.9,A -85,B 0,C 180,E1 17200.328,E2 17200.328} C_VEL
LIN {X 0,Y 495.969,Z 1276.996,A -85,B 0,C 180,E1 17197.643,E2 17197.643} C_VEL
LIN {X 0,Y 495.92,Z 1280.196,A -85,B 0,C 180,E1 17194.622,E2 17194.622} C_VEL
LIN {X 0,Y 495.906,Z 1281.69,A -85,B 0,C 180,E1 17191.614,E2 17191.614} C_VEL
LIN {X 0,Y 495.866,Z 1281.848,A -85,B 0,C 180,E1 17189.188,E2 17189.188} C_VEL
LIN {X 0,Y 495.911,Z 1281.011,A -85,B 0,C 180,E1 17186.76,E2 17186.76} C_VEL
LIN {X 0,Y 495.935,Z 1279.19,A -85,B 0,C 180,E1 17184.327,E2 17184.327} C_VEL
LIN {X 0,Y 495.99,Z 1276.346,A -85,B 0,C 180,E1 17181.885,E2 17181.885} C_VEL
LIN {X 0,Y 496.202,Z 1272.268,A -85,B 0,C 180,E1 17179.313,E2 17179.313} C_VEL
LIN {X 0,Y 496.62,Z 1266.52,A -85,B 0,C 180,E1 17176.491,E2 17176.491} C_VEL
LIN {X 0,Y 497.463,Z 1258.257,A -85,B 0,C 180,E1 17173.293,E2 17173.293} C_VEL
LIN {X 0,Y 498.516,Z 1250.089,A -85,B 0,C 180,E1 17170.671,E2 17170.671} C_VEL
LIN {X 0,Y 499.887,Z 1241.505,A -85,B 0,C 180,E1 17168.279,E2 17168.279} C_VEL
LIN {X 0,Y 501.651,Z 1231.728,A -85,B 0,C 180,E1 17165.88,E2 17165.88} C_VEL
LIN {X 0,Y 504.16,Z 1219.211,A -85,B 0,C 180,E1 17163.187,E2 17163.187} C_VEL
LIN {X 0,Y 507.47,Z 1203.85,A -85,B 0,C 180,E1 17160.334,E2 17160.334} C_VEL
LIN {X 0,Y 510.673,Z 1190.091,A -85,B 0,C 180,E1 17158.083,E2 17158.083} C_VEL
LIN {X 0,Y 514.004,Z 1176.311,A -85,B 0,C 180,E1 17156.06,E2 17156.06} C_VEL
LIN {X 0,Y 517.847,Z 1160.714,A -85,B 0,C 180,E1 17154.002,E2 17154.002} C_VEL
LIN {X 0,Y 523.031,Z 1139.946,A -85,B 0,C 180,E1 17151.586,E2 17151.586} C_VEL
LIN {X 0,Y 527.683,Z 1121.019,A -85,B 0,C 180,E1 17149.675,E2 17149.675} C_VEL
LIN {X 0,Y 531.983,Z 1103.178,A -85,B 0,C 180,E1 17148.072,E2 17148.072} C_VEL
LIN {X 0,Y 536.45,Z 1084.055,A -85,B 0,C 180,E1 17146.544,E2 17146.544} C_VEL
LIN {X 0,Y 541.809,Z 1060.061,A -85,B 0,C 180,E1 17144.873,E2 17144.873} C_VEL
LIN {X 0,Y 546.318,Z 1037.761,A -85,B 0,C 180,E1 17143.549,E2 17143.549} C_VEL
LIN {X 0,Y 550.062,Z 1017.717,A -85,B 0,C 180,E1 17142.513,E2 17142.513} C_VEL
LIN {X 0,Y 553.358,Z 998.523,A -85,B 0,C 180,E1 17141.653,E2 17141.653} C_VEL
LIN {X 0,Y 556.549,Z 977.786,A -85,B 0,C 180,E1 17140.854,E2 17140.854} C_VEL
LIN {X 0,Y 559.495,Z 955.854,A -85,B 0,C 180,E1 17140.146,E2 17140.146} C_VEL
LIN {X 0,Y 562.642,Z 927.208,A -85,B 0,C 180,E1 17139.42,E2 17139.42} C_VEL
LIN {X 0,Y 564.573,Z 902.637,A -85,B 0,C 180,E1 17138.963,E2 17138.963} C_VEL
LIN {X 0,Y 573.015,Z 704.424,A -85,B 0,C 180,E1 17136.004,E2 17136.004} C_VEL
LIN {X 0,Y 580.48,Z 534.967,A -85,B 0,C 180,E1 17133.45,E2 17133.45} C_VEL
LIN {X 0,Y 569.141,Z 517.508,A -85,B 0,C 180,E1 17131.275,E2 17131.275} C_VEL
LIN {X 0,Y 557.708,Z 500.96,A -85,B 0,C 180,E1 17128.864,E2 17128.864} C_VEL
LIN {X 0,Y 548.236,Z 488.13,A -85,B 0,C 180,E1 17126.658,E2 17126.658} C_VEL
LIN {X 0,Y 540.55,Z 478.04,A -85,B 0,C 180,E1 17124.682,E2 17124.682} C_VEL
LIN {X 0,Y 536.667,Z 473.297,A -85,B 0,C 180,E1 17123.614,E2 17123.614} C_VEL
LIN {X 0,Y 532.962,Z 468.651,A -85,B 0,C 180,E1 17122.532,E2 17122.532} C_VEL
LIN {X 0,Y 528.704,Z 464.139,A -85,B 0,C 180,E1 17121.233,E2 17121.233} C_VEL
LIN {X 0,Y 527.159,Z 461.932,A -85,B 0,C 180,E1 17120.717,E2 17120.717} C_VEL
LIN {X 0,Y 523.664,Z 458.508,A -85,B 0,C 180,E1 17119.55,E2 17119.55} C_VEL
LIN {X 0,Y 521.911,Z 455.794,A -85,B 0,C 180,E1 17118.891,E2 17118.891} C_VEL
LIN {X 0,Y 518.601,Z 453.077,A -85,B 0,C 180,E1 17117.678,E2 17117.678} C_VEL
LIN {X 0,Y 516.492,Z 449.488,A -85,B 0,C 180,E1 17116.765,E2 17116.765} C_VEL
LIN {X 0,Y 513.146,Z 447.17,A -85,B 0,C 180,E1 17115.367,E2 17115.367} C_VEL
LIN {X 0,Y 510.965,Z 443.855,A -85,B 0,C 180,E1 17114.274,E2 17114.274} C_VEL
LIN {X 0,Y 510.362,Z 442.738,A -85,B 0,C 180,E1 17113.944,E2 17113.944} C_VEL
LIN {X 0,Y 506.953,Z 440.78,A -85,B 0,C 180,E1 17112.183,E2 17112.183} C_VEL
LIN {X 0,Y 504.845,Z 437.435,A -85,B 0,C 180,E1 17110.787,E2 17110.787} C_VEL
LIN {X 0,Y 504.365,Z 436.035,A -85,B 0,C 180,E1 17110.393,E2 17110.393} C_VEL
LIN {X 0,Y 500.4,Z 434.01,A -85,B 0,C 180,E1 17107.347,E2 17107.347} C_VEL
LIN {X 0,Y 498.257,Z 430.762,A -85,B 0,C 180,E1 17104.604,E2 17104.604} C_VEL
LIN {X 0,Y 497.916,Z 429.136,A -85,B 0,C 180,E1 17103.684,E2 17103.684} C_VEL
LIN {X 0,Y 497.903,Z 429.211,A -85,B 0,C 180,E1 17100.115,E2 17100.115} C_VEL
LIN {X 0,Y 497.897,Z 429.136,A -85,B 0,C 180,E1 17096.465,E2 17096.465} C_VEL
LIN {X 0,Y 497.945,Z 429.451,A -85,B 0,C 180,E1 17095.912,E2 17095.912} C_VEL
LIN {X 0,Y 499.371,Z 432.883,A -85,B 0,C 180,E1 17093.562,E2 17093.562} C_VEL
LIN {X 0,Y 503.062,Z 435.653,A -85,B 0,C 180,E1 17090.273,E2 17090.273} C_VEL
LIN {X 0,Y 504.524,Z 436.278,A -85,B 0,C 180,E1 17089.292,E2 17089.292} C_VEL
LIN {X 0,Y 505.832,Z 439.401,A -85,B 0,C 180,E1 17088.31,E2 17088.31} C_VEL
LIN {X 0,Y 508.634,Z 441.991,A -85,B 0,C 180,E1 17086.703,E2 17086.703} C_VEL
LIN {X 0,Y 510.698,Z 443.052,A -85,B 0,C 180,E1 17085.689,E2 17085.689} C_VEL
LIN {X 0,Y 512.628,Z 446.594,A -85,B 0,C 180,E1 17084.675,E2 17084.675} C_VEL
LIN {X 0,Y 515.753,Z 449.131,A -85,B 0,C 180,E1 17083.326,E2 17083.326} C_VEL
LIN {X 0,Y 516.686,Z 449.903,A -85,B 0,C 180,E1 17082.945,E2 17082.945} C_VEL
LIN {X 0,Y 519.09,Z 453.583,A -85,B 0,C 180,E1 17081.933,E2 17081.933} C_VEL
LIN {X 0,Y 522.358,Z 456.271,A -85,B 0,C 180,E1 17080.748,E2 17080.748} C_VEL
LIN {X 0,Y 525.178,Z 460.25,A -85,B 0,C 180,E1 17079.726,E2 17079.726} C_VEL
LIN {X 0,Y 527.885,Z 462.736,A -85,B 0,C 180,E1 17078.848,E2 17078.848} C_VEL
LIN {X 0,Y 531.255,Z 467.063,A -85,B 0,C 180,E1 17077.771,E2 17077.771} C_VEL
LIN {X 0,Y 533.227,Z 469.004,A -85,B 0,C 180,E1 17077.189,E2 17077.189} C_VEL
LIN {X 0,Y 536.957,Z 473.511,A -85,B 0,C 180,E1 17076.109,E2 17076.109} C_VEL
LIN {X 0,Y 539.199,Z 476.332,A -85,B 0,C 180,E1 17075.485,E2 17075.485} C_VEL
LIN {X 0,Y 543.393,Z 481.309,A -85,B 0,C 180,E1 17074.379,E2 17074.379} C_VEL
LIN {X 0,Y 548.631,Z 487.826,A -85,B 0,C 180,E1 17073.07,E2 17073.07} C_VEL
LIN {X 0,Y 553.49,Z 493.908,A -85,B 0,C 180,E1 17071.927,E2 17071.927} C_VEL
LIN {X 0,Y 563.742,Z 507.126,A -85,B 0,C 180,E1 17069.694,E2 17069.694} C_VEL
LIN {X 0,Y 572.94,Z 520.467,A -85,B 0,C 180,E1 17067.84,E2 17067.84} C_VEL
LIN {X 0,Y 580.491,Z 532.068,A -85,B 0,C 180,E1 17066.413,E2 17066.413} C_VEL
LIN {X 0,Y 571.022,Z 747.026,A -85,B 0,C 180,E1 17063.185,E2 17063.185} C_VEL
LIN {X 0,Y 564.67,Z 895.278,A -85,B 0,C 180,E1 17060.97,E2 17060.97} C_VEL
LIN {X 0,Y 562.649,Z 921.058,A -85,B 0,C 180,E1 17060.482,E2 17060.482} C_VEL
LIN {X 0,Y 559.603,Z 948.488,A -85,B 0,C 180,E1 17059.771,E2 17059.771} C_VEL
LIN {X 0,Y 556.761,Z 969.708,A -85,B 0,C 180,E1 17059.081,E2 17059.081} C_VEL
LIN {X 0,Y 553.7,Z 989.728,A -85,B 0,C 180,E1 17058.308,E2 17058.308} C_VEL
LIN {X 0,Y 550.21,Z 1010.047,A -85,B 0,C 180,E1 17057.393,E2 17057.393} C_VEL
LIN {X 0,Y 545.9,Z 1032.934,A -85,B 0,C 180,E1 17056.194,E2 17056.194} C_VEL
LIN {X 0,Y 540.668,Z 1057.813,A -85,B 0,C 180,E1 17054.65,E2 17054.65} C_VEL
LIN {X 0,Y 539.639,Z 1062.49,A -85,B 0,C 180,E1 17054.327,E2 17054.327} C_VEL
LIN {X 0,Y 537.483,Z 1069.152,A -85,B 0,C 180,E1 17053.942,E2 17053.942} C_VEL
LIN {X 0,Y 528.712,Z 1086.625,A -85,B 0,C 180,E1 17053.083,E2 17053.083} C_VEL
LIN {X 0,Y 526.772,Z 1091.882,A -85,B 0,C 180,E1 17052.696,E2 17052.696} C_VEL
LIN {X 0,Y 522.315,Z 1109.503,A -85,B 0,C 180,E1 17051.117,E2 17051.117} C_VEL
LIN {X 0,Y 518.239,Z 1125.192,A -85,B 0,C 180,E1 17049.548,E2 17049.548} C_VEL
LIN {X 0,Y 514.063,Z 1141.014,A -85,B 0,C 180,E1 17047.787,E2 17047.787} C_VEL
LIN {X 0,Y 509.778,Z 1157.222,A -85,B 0,C 180,E1 17045.77,E2 17045.77} C_VEL
LIN {X 0,Y 504.697,Z 1176.613,A -85,B 0,C 180,E1 17043.015,E2 17043.015} C_VEL
LIN {X 0,Y 501.099,Z 1190.906,A -85,B 0,C 180,E1 17040.681,E2 17040.681} C_VEL
LIN {X 0,Y 498.108,Z 1203.327,A -85,B 0,C 180,E1 17038.41,E2 17038.41} C_VEL
LIN {X 0,Y 495.414,Z 1215.193,A -85,B 0,C 180,E1 17035.977,E2 17035.977} C_VEL
LIN {X 0,Y 492.767,Z 1228.306,A -85,B 0,C 180,E1 17032.893,E2 17032.893} C_VEL
LIN {X 0,Y 490.93,Z 1238.727,A -85,B 0,C 180,E1 17030.012,E2 17030.012} C_VEL
LIN {X 0,Y 489.794,Z 1246.421,A -85,B 0,C 180,E1 17027.567,E2 17027.567} C_VEL
LIN {X 0,Y 489.023,Z 1252.922,A -85,B 0,C 180,E1 17025.175,E2 17025.175} C_VEL
LIN {X 0,Y 488.46,Z 1258.713,A -85,B 0,C 180,E1 17022.655,E2 17022.655} C_VEL
LIN {X 0,Y 488.12,Z 1263.633,A -85,B 0,C 180,E1 17020.03,E2 17020.03} C_VEL
LIN {X 0,Y 487.964,Z 1268.12,A -85,B 0,C 180,E1 17016.829,E2 17016.829} C_VEL
LIN {X 0,Y 487.916,Z 1270.645,A -85,B 0,C 180,E1 17013.881,E2 17013.881} C_VEL
LIN {X 0,Y 487.903,Z 1271.725,A -85,B 0,C 180,E1 17011.412,E2 17011.412} C_VEL
LIN {X 0,Y 487.87,Z 1271.835,A -85,B 0,C 180,E1 17009.064,E2 17009.064} C_VEL
LIN {X 0,Y 487.911,Z 1271.042,A -85,B 0,C 180,E1 17006.714,E2 17006.714} C_VEL
LIN {X 0,Y 487.937,Z 1269.238,A -85,B 0,C 180,E1 17004.241,E2 17004.241} C_VEL
LIN {X 0,Y 488.005,Z 1266.399,A -85,B 0,C 180,E1 17001.746,E2 17001.746} C_VEL
LIN {X 0,Y 488.215,Z 1262.355,A -85,B 0,C 180,E1 16999.143,E2 16999.143} C_VEL
LIN {X 0,Y 488.639,Z 1256.883,A -85,B 0,C 180,E1 16996.394,E2 16996.394} C_VEL
LIN {X 0,Y 489.563,Z 1248.408,A -85,B 0,C 180,E1 16993.023,E2 16993.023} C_VEL
LIN {X 0,Y 490.678,Z 1240.26,A -85,B 0,C 180,E1 16990.357,E2 16990.357} C_VEL
LIN {X 0,Y 492.153,Z 1231.555,A -85,B 0,C 180,E1 16987.887,E2 16987.887} C_VEL
LIN {X 0,Y 493.998,Z 1222.014,A -85,B 0,C 180,E1 16985.49,E2 16985.49} C_VEL
LIN {X 0,Y 496.612,Z 1209.924,A -85,B 0,C 180,E1 16982.808,E2 16982.808} C_VEL
LIN {X 0,Y 500.172,Z 1194.692,A -85,B 0,C 180,E1 16979.888,E2 16979.888} C_VEL
LIN {X 0,Y 503.655,Z 1180.686,A -85,B 0,C 180,E1 16977.538,E2 16977.538} C_VEL
LIN {X 0,Y 507.314,Z 1166.555,A -85,B 0,C 180,E1 16975.421,E2 16975.421} C_VEL
LIN {X 0,Y 511.569,Z 1150.428,A -85,B 0,C 180,E1 16973.261,E2 16973.261} C_VEL
LIN {X 0,Y 517.168,Z 1129.269,A -85,B 0,C 180,E1 16970.792,E2 16970.792} C_VEL
LIN {X 0,Y 521.788,Z 1111.533,A -85,B 0,C 180,E1 16968.985,E2 16968.985} C_VEL
LIN {X 0,Y 526.125,Z 1094.437,A -85,B 0,C 180,E1 16967.431,E2 16967.431} C_VEL
LIN {X 0,Y 530.783,Z 1075.433,A -85,B 0,C 180,E1 16965.895,E2 16965.895} C_VEL
LIN {X 0,Y 536.404,Z 1051.281,A -85,B 0,C 180,E1 16964.2,E2 16964.2} C_VEL
LIN {X 0,Y 541.022,Z 1029.328,A -85,B 0,C 180,E1 16962.887,E2 16962.887} C_VEL
LIN {X 0,Y 544.892,Z 1009.353,A -85,B 0,C 180,E1 16961.847,E2 16961.847} C_VEL
LIN {X 0,Y 548.289,Z 990.203,A -85,B 0,C 180,E1 16960.983,E2 16960.983} C_VEL
LIN {X 0,Y 551.489,Z 970.019,A -85,B 0,C 180,E1 16960.2,E2 16960.2} C_VEL
LIN {X 0,Y 554.503,Z 948.203,A -85,B 0,C 180,E1 16959.489,E2 16959.489} C_VEL
LIN {X 0,Y 557.684,Z 920.037,A -85,B 0,C 180,E1 16958.765,E2 16958.765} C_VEL
LIN {X 0,Y 559.694,Z 895.099,A -85,B 0,C 180,E1 16958.295,E2 16958.295} C_VEL
LIN {X 0,Y 567.509,Z 719.484,A -85,B 0,C 180,E1 16955.658,E2 16955.658} C_VEL
LIN {X 0,Y 575.927,Z 536.174,A -85,B 0,C 180,E1 16952.887,E2 16952.887} C_VEL
LIN {X 0,Y 563.909,Z 518.128,A -85,B 0,C 180,E1 16950.502,E2 16950.502} C_VEL
LIN {X 0,Y 556.037,Z 507.416,A -85,B 0,C 180,E1 16948.812,E2 16948.812} C_VEL
LIN {X 0,Y 547.447,Z 496.44,A -85,B 0,C 180,E1 16946.817,E2 16946.817} C_VEL
LIN {X 0,Y 542.698,Z 490.507,A -85,B 0,C 180,E1 16945.627,E2 16945.627} C_VEL
LIN {X 0,Y 539.249,Z 486.21,A -85,B 0,C 180,E1 16944.717,E2 16944.717} C_VEL
LIN {X 0,Y 534.946,Z 480.941,A -85,B 0,C 180,E1 16943.52,E2 16943.52} C_VEL
LIN {X 0,Y 531.023,Z 476.094,A -85,B 0,C 180,E1 16942.356,E2 16942.356} C_VEL
LIN {X 0,Y 526.683,Z 471.337,A -85,B 0,C 180,E1 16940.998,E2 16940.998} C_VEL
LIN {X 0,Y 525.229,Z 469.379,A -85,B 0,C 180,E1 16940.505,E2 16940.505} C_VEL
LIN {X 0,Y 521.743,Z 465.754,A -85,B 0,C 180,E1 16939.304,E2 16939.304} C_VEL
LIN {X 0,Y 520.226,Z 463.428,A -85,B 0,C 180,E1 16938.722,E2 16938.722} C_VEL
LIN {X 0,Y 516.855,Z 460.48,A -85,B 0,C 180,E1 16937.449,E2 16937.449} C_VEL
LIN {X 0,Y 514.904,Z 457.219,A -85,B 0,C 180,E1 16936.586,E2 16936.586} C_VEL
LIN {X 0,Y 511.53,Z 454.66,A -85,B 0,C 180,E1 16935.127,E2 16935.127} C_VEL
LIN {X 0,Y 509.321,Z 451.132,A -85,B 0,C 180,E1 16933.973,E2 16933.973} C_VEL
LIN {X 0,Y 508.915,Z 450.538,A -85,B 0,C 180,E1 16933.753,E2 16933.753} C_VEL
LIN {X 0,Y 505.427,Z 448.307,A -85,B 0,C 180,E1 16931.873,E2 16931.873} C_VEL
LIN {X 0,Y 503.362,Z 444.693,A -85,B 0,C 180,E1 16930.414,E2 16930.414} C_VEL
LIN {X 0,Y 502.93,Z 443.881,A -85,B 0,C 180,E1 16930.076,E2 16930.076} C_VEL
LIN {X 0,Y 498.873,Z 441.523,A -85,B 0,C 180,E1 16926.676,E2 16926.676} C_VEL
LIN {X 0,Y 496.952,Z 437.705,A -85,B 0,C 180,E1 16923.576,E2 16923.576} C_VEL
LIN {X 0,Y 496.802,Z 437.058,A -85,B 0,C 180,E1 16923.115,E2 16923.115} C_VEL
LIN {X 0,Y 496.88,Z 437.296,A -85,B 0,C 180,E1 16916.77,E2 16916.77} C_VEL
LIN {X 0,Y 498.473,Z 441.098,A -85,B 0,C 180,E1 16913.897,E2 16913.897} C_VEL
LIN {X 0,Y 502.265,Z 443.671,A -85,B 0,C 180,E1 16910.489,E2 16910.489} C_VEL
LIN {X 0,Y 503.225,Z 444.26,A -85,B 0,C 180,E1 16909.814,E2 16909.814} C_VEL
LIN {X 0,Y 505.147,Z 448.002,A -85,B 0,C 180,E1 16908.41,E2 16908.41} C_VEL
LIN {X 0,Y 508.23,Z 450.279,A -85,B 0,C 180,E1 16906.692,E2 16906.692} C_VEL
LIN {X 0,Y 509.263,Z 450.997,A -85,B 0,C 180,E1 16906.17,E2 16906.17} C_VEL
LIN {X 0,Y 511.514,Z 454.664,A -85,B 0,C 180,E1 16904.989,E2 16904.989} C_VEL
LIN {X 0,Y 515.059,Z 457.571,A -85,B 0,C 180,E1 16903.448,E2 16903.448} C_VEL
LIN {X 0,Y 517.632,Z 461.418,A -85,B 0,C 180,E1 16902.346,E2 16902.346} C_VEL
LIN {X 0,Y 520.625,Z 463.963,A -85,B 0,C 180,E1 16901.235,E2 16901.235} C_VEL
LIN {X 0,Y 523.79,Z 468.179,A -85,B 0,C 180,E1 16900.077,E2 16900.077} C_VEL
LIN {X 0,Y 525.985,Z 470.25,A -85,B 0,C 180,E1 16899.351,E2 16899.351} C_VEL
LIN {X 0,Y 529.47,Z 474.666,A -85,B 0,C 180,E1 16898.217,E2 16898.217} C_VEL
LIN {X 0,Y 531.4,Z 476.737,A -85,B 0,C 180,E1 16897.632,E2 16897.632} C_VEL
LIN {X 0,Y 536.771,Z 483.257,A -85,B 0,C 180,E1 16896.07,E2 16896.07} C_VEL
LIN {X 0,Y 543.468,Z 492.086,A -85,B 0,C 180,E1 16894.265,E2 16894.265} C_VEL
LIN {X 0,Y 550.809,Z 501.953,A -85,B 0,C 180,E1 16892.454,E2 16892.454} C_VEL
LIN {X 0,Y 560.49,Z 515.715,A -85,B 0,C 180,E1 16890.268,E2 16890.268} C_VEL
LIN {X 0,Y 570.672,Z 530.965,A -85,B 0,C 180,E1 16888.171,E2 16888.171} C_VEL
LIN {X 0,Y 575.947,Z 539.621,A -85,B 0,C 180,E1 16887.142,E2 16887.142} C_VEL
LIN {X 0,Y 565.999,Z 757.523,A -85,B 0,C 180,E1 16883.857,E2 16883.857} C_VEL
LIN {X 0,Y 559.557,Z 902.87,A -85,B 0,C 180,E1 16881.674,E2 16881.674} C_VEL
LIN {X 0,Y 557.438,Z 928.854,A -85,B 0,C 180,E1 16881.185,E2 16881.185} C_VEL
LIN {X 0,Y 554.255,Z 956.382,A -85,B 0,C 180,E1 16880.475,E2 16880.475} C_VEL
LIN {X 0,Y 551.26,Z 977.934,A -85,B 0,C 180,E1 16879.777,E2 16879.777} C_VEL
LIN {X 0,Y 547.96,Z 998.633,A -85,B 0,C 180,E1 16878.977,E2 16878.977} C_VEL
LIN {X 0,Y 544.224,Z 1019.594,A -85,B 0,C 180,E1 16878.028,E2 16878.028} C_VEL
LIN {X 0,Y 539.256,Z 1044.886,A -85,B 0,C 180,E1 16876.681,E2 16876.681} C_VEL
LIN {X 0,Y 534.282,Z 1067.47,A -85,B 0,C 180,E1 16875.253,E2 16875.253} C_VEL
LIN {X 0,Y 529.727,Z 1087.019,A -85,B 0,C 180,E1 16873.84,E2 16873.84} C_VEL
LIN {X 0,Y 525.138,Z 1105.859,A -85,B 0,C 180,E1 16872.299,E2 16872.299} C_VEL
LIN {X 0,Y 519.539,Z 1128.115,A -85,B 0,C 180,E1 16870.224,E2 16870.224} C_VEL
LIN {X 0,Y 514.558,Z 1147.224,A -85,B 0,C 180,E1 16868.159,E2 16868.159} C_VEL
LIN {X 0,Y 510.469,Z 1162.899,A -85,B 0,C 180,E1 16866.261,E2 16866.261} C_VEL
LIN {X 0,Y 506.595,Z 1177.968,A -85,B 0,C 180,E1 16864.224,E2 16864.224} C_VEL
LIN {X 0,Y 502.414,Z 1194.693,A -85,B 0,C 180,E1 16861.69,E2 16861.69} C_VEL
LIN {X 0,Y 498.564,Z 1210.606,A -85,B 0,C 180,E1 16858.898,E2 16858.898} C_VEL
LIN {X 0,Y 495.821,Z 1222.855,A -85,B 0,C 180,E1 16856.461,E2 16856.461} C_VEL
LIN {X 0,Y 493.607,Z 1233.743,A -85,B 0,C 180,E1 16854.022,E2 16854.022} C_VEL
LIN {X 0,Y 491.562,Z 1245.197,A -85,B 0,C 180,E1 16851.098,E2 16851.098} C_VEL
LIN {X 0,Y 489.933,Z 1255.453,A -85,B 0,C 180,E1 16847.945,E2 16847.945} C_VEL
LIN {X 0,Y 489.085,Z 1262.448,A -85,B 0,C 180,E1 16845.409,E2 16845.409} C_VEL
LIN {X 0,Y 488.499,Z 1268.314,A -85,B 0,C 180,E1 16842.888,E2 16842.888} C_VEL
LIN {X 0,Y 488.169,Z 1273.103,A -85,B 0,C 180,E1 16840.38,E2 16840.38} C_VEL
LIN {X 0,Y 487.972,Z 1277.312,A -85,B 0,C 180,E1 16837.532,E2 16837.532} C_VEL
LIN {X 0,Y 487.92,Z 1280.403,A -85,B 0,C 180,E1 16834.345,E2 16834.345} C_VEL
LIN {X 0,Y 487.906,Z 1281.69,A -85,B 0,C 180,E1 16831.641,E2 16831.641} C_VEL
LIN {X 0,Y 487.867,Z 1281.847,A -85,B 0,C 180,E1 16829.175,E2 16829.175} C_VEL
LIN {X 0,Y 487.912,Z 1281.011,A -85,B 0,C 180,E1 16826.707,E2 16826.707} C_VEL
LIN {X 0,Y 487.938,Z 1279.187,A -85,B 0,C 180,E1 16824.234,E2 16824.234} C_VEL
LIN {X 0,Y 488.006,Z 1276.335,A -85,B 0,C 180,E1 16821.745,E2 16821.745} C_VEL
LIN {X 0,Y 488.221,Z 1272.265,A -85,B 0,C 180,E1 16819.137,E2 16819.137} C_VEL
LIN {X 0,Y 488.646,Z 1266.774,A -85,B 0,C 180,E1 16816.387,E2 16816.387} C_VEL
LIN {X 0,Y 489.539,Z 1258.609,A -85,B 0,C 180,E1 16813.137,E2 16813.137} C_VEL
LIN {X 0,Y 490.643,Z 1250.493,A -85,B 0,C 180,E1 16810.472,E2 16810.472} C_VEL
LIN {X 0,Y 492.08,Z 1241.957,A -85,B 0,C 180,E1 16808.042,E2 16808.042} C_VEL
LIN {X 0,Y 493.92,Z 1232.165,A -85,B 0,C 180,E1 16805.606,E2 16805.606} C_VEL
LIN {X 0,Y 496.356,Z 1220.519,A -85,B 0,C 180,E1 16803.045,E2 16803.045} C_VEL
LIN {X 0,Y 500.158,Z 1203.885,A -85,B 0,C 180,E1 16799.88,E2 16799.88} C_VEL
LIN {X 0,Y 503.57,Z 1189.851,A -85,B 0,C 180,E1 16797.553,E2 16797.553} C_VEL
LIN {X 0,Y 507.052,Z 1176.138,A -85,B 0,C 180,E1 16795.516,E2 16795.516} C_VEL
LIN {X 0,Y 511.065,Z 1160.614,A -85,B 0,C 180,E1 16793.446,E2 16793.446} C_VEL
LIN {X 0,Y 516.496,Z 1139.853,A -85,B 0,C 180,E1 16791.009,E2 16791.009} C_VEL
LIN {X 0,Y 521.353,Z 1120.925,A -85,B 0,C 180,E1 16789.082,E2 16789.082} C_VEL
LIN {X 0,Y 525.657,Z 1103.754,A -85,B 0,C 180,E1 16787.523,E2 16787.523} C_VEL
LIN {X 0,Y 530.104,Z 1085.435,A -85,B 0,C 180,E1 16786.041,E2 16786.041} C_VEL
LIN {X 0,Y 535.251,Z 1063.363,A -85,B 0,C 180,E1 16784.469,E2 16784.469} C_VEL
LIN {X 0,Y 540.5,Z 1038.674,A -85,B 0,C 180,E1 16782.974,E2 16782.974} C_VEL
LIN {X 0,Y 544.573,Z 1017.622,A -85,B 0,C 180,E1 16781.879,E2 16781.879} C_VEL
LIN {X 0,Y 547.977,Z 998.426,A -85,B 0,C 180,E1 16781.016,E2 16781.016} C_VEL
LIN {X 0,Y 551.278,Z 977.689,A -85,B 0,C 180,E1 16780.216,E2 16780.216} C_VEL
LIN {X 0,Y 554.322,Z 955.734,A -85,B 0,C 180,E1 16779.507,E2 16779.507} C_VEL
LIN {X 0,Y 557.566,Z 927.106,A -85,B 0,C 180,E1 16778.781,E2 16778.781} C_VEL
LIN {X 0,Y 559.553,Z 902.525,A -85,B 0,C 180,E1 16778.323,E2 16778.323} C_VEL
LIN {X 0,Y 568.453,Z 701.369,A -85,B 0,C 180,E1 16775.303,E2 16775.303} C_VEL
LIN {X 0,Y 575.865,Z 539.206,A -85,B 0,C 180,E1 16772.846,E2 16772.846} C_VEL
LIN {X 0,Y 565.67,Z 523.464,A -85,B 0,C 180,E1 16770.838,E2 16770.838} C_VEL
LIN {X 0,Y 554.936,Z 507.69,A -85,B 0,C 180,E1 16768.521,E2 16768.521} C_VEL
LIN {X 0,Y 545.687,Z 495.037,A -85,B 0,C 180,E1 16766.323,E2 16766.323} C_VEL
LIN {X 0,Y 538.201,Z 485.083,A -85,B 0,C 180,E1 16764.358,E2 16764.358} C_VEL
LIN {X 0,Y 534.637,Z 480.667,A -85,B 0,C 180,E1 16763.359,E2 16763.359} C_VEL
LIN {X 0,Y 530.206,Z 475.313,A -85,B 0,C 180,E1 16762.042,E2 16762.042} C_VEL
LIN {X 0,Y 526.503,Z 471.099,A -85,B 0,C 180,E1 16760.873,E2 16760.873} C_VEL
LIN {X 0,Y 525.242,Z 469.396,A -85,B 0,C 180,E1 16760.446,E2 16760.446} C_VEL
LIN {X 0,Y 521.739,Z 465.766,A -85,B 0,C 180,E1 16759.246,E2 16759.246} C_VEL
LIN {X 0,Y 520.065,Z 463.339,A -85,B 0,C 180,E1 16758.612,E2 16758.612} C_VEL
LIN {X 0,Y 516.699,Z 460.279,A -85,B 0,C 180,E1 16757.338,E2 16757.338} C_VEL
LIN {X 0,Y 514.73,Z 457.13,A -85,B 0,C 180,E1 16756.476,E2 16756.476} C_VEL
LIN {X 0,Y 511.358,Z 454.47,A -85,B 0,C 180,E1 16755.016,E2 16755.016} C_VEL
LIN {X 0,Y 509.21,Z 450.88,A -85,B 0,C 180,E1 16753.89,E2 16753.89} C_VEL
LIN {X 0,Y 505.24,Z 448.074,A -85,B 0,C 180,E1 16751.762,E2 16751.762} C_VEL
LIN {X 0,Y 503.297,Z 444.503,A -85,B 0,C 180,E1 16750.387,E2 16750.387} C_VEL
LIN {X 0,Y 503.054,Z 443.901,A -85,B 0,C 180,E1 16750.189,E2 16750.189} C_VEL
LIN {X 0,Y 499.084,Z 441.696,A -85,B 0,C 180,E1 16747.02,E2 16747.02} C_VEL
LIN {X 0,Y 497.022,Z 437.997,A -85,B 0,C 180,E1 16744.095,E2 16744.095} C_VEL
LIN {X 0,Y 496.766,Z 437.048,A -85,B 0,C 180,E1 16743.462,E2 16743.462} C_VEL
LIN {X 0,Y 496.868,Z 437.142,A -85,B 0,C 180,E1 16736.134,E2 16736.134} C_VEL
LIN {X 0,Y 498.3,Z 440.761,A -85,B 0,C 180,E1 16733.664,E2 16733.664} C_VEL
LIN {X 0,Y 501.941,Z 443.546,A -85,B 0,C 180,E1 16730.367,E2 16730.367} C_VEL
LIN {X 0,Y 503.213,Z 444.123,A -85,B 0,C 180,E1 16729.496,E2 16729.496} C_VEL
LIN {X 0,Y 504.763,Z 447.461,A -85,B 0,C 180,E1 16728.343,E2 16728.343} C_VEL
LIN {X 0,Y 507.894,Z 450.102,A -85,B 0,C 180,E1 16726.567,E2 16726.567} C_VEL
LIN {X 0,Y 509.273,Z 450.93,A -85,B 0,C 180,E1 16725.88,E2 16725.88} C_VEL
LIN {X 0,Y 511.537,Z 454.695,A -85,B 0,C 180,E1 16724.699,E2 16724.699} C_VEL
LIN {X 0,Y 515.053,Z 457.516,A -85,B 0,C 180,E1 16723.186,E2 16723.186} C_VEL
LIN {X 0,Y 517.714,Z 461.42,A -85,B 0,C 180,E1 16722.058,E2 16722.058} C_VEL
LIN {X 0,Y 520.723,Z 464.038,A -85,B 0,C 180,E1 16720.947,E2 16720.947} C_VEL
LIN {X 0,Y 523.913,Z 468.249,A -85,B 0,C 180,E1 16719.791,E2 16719.791} C_VEL
LIN {X 0,Y 526.04,Z 470.261,A -85,B 0,C 180,E1 16719.092,E2 16719.092} C_VEL
LIN {X 0,Y 529.459,Z 474.607,A -85,B 0,C 180,E1 16717.984,E2 16717.984} C_VEL
LIN {X 0,Y 531.318,Z 476.529,A -85,B 0,C 180,E1 16717.424,E2 16717.424} C_VEL
LIN {X 0,Y 535.292,Z 481.224,A -85,B 0,C 180,E1 16716.263,E2 16716.263} C_VEL
LIN {X 0,Y 541.471,Z 488.971,A -85,B 0,C 180,E1 16714.574,E2 16714.574} C_VEL
LIN {X 0,Y 546.57,Z 495.35,A -85,B 0,C 180,E1 16713.284,E2 16713.284} C_VEL
LIN {X 0,Y 553.455,Z 504.034,A -85,B 0,C 180,E1 16711.66,E2 16711.66} C_VEL
LIN {X 0,Y 563.41,Z 517.402,A -85,B 0,C 180,E1 16709.498,E2 16709.498} C_VEL
LIN {X 0,Y 575.296,Z 535.241,A -85,B 0,C 180,E1 16707.132,E2 16707.132} C_VEL
LIN {X 0,Y 575.885,Z 536.487,A -85,B 0,C 180,E1 16707.013,E2 16707.013} C_VEL
LIN {X 0,Y 566.027,Z 752.242,A -85,B 0,C 180,E1 16703.758,E2 16703.758} C_VEL
LIN {X 0,Y 559.654,Z 895.391,A -85,B 0,C 180,E1 16701.608,E2 16701.608} C_VEL
LIN {X 0,Y 557.563,Z 921.266,A -85,B 0,C 180,E1 16701.117,E2 16701.117} C_VEL
LIN {X 0,Y 554.432,Z 948.589,A -85,B 0,C 180,E1 16700.407,E2 16700.407} C_VEL
LIN {X 0,Y 551.501,Z 969.807,A -85,B 0,C 180,E1 16699.716,E2 16699.716} C_VEL
LIN {X 0,Y 548.338,Z 989.826,A -85,B 0,C 180,E1 16698.941,E2 16698.941} C_VEL
LIN {X 0,Y 544.733,Z 1010.145,A -85,B 0,C 180,E1 16698.023,E2 16698.023} C_VEL
LIN {X 0,Y 540.471,Z 1032.03,A -85,B 0,C 180,E1 16696.874,E2 16696.874} C_VEL
LIN {X 0,Y 534.852,Z 1057.91,A -85,B 0,C 180,E1 16695.269,E2 16695.269} C_VEL
LIN {X 0,Y 530.108,Z 1078.105,A -85,B 0,C 180,E1 16693.809,E2 16693.809} C_VEL
LIN {X 0,Y 526.772,Z 1091.882,A -85,B 0,C 180,E1 16692.696,E2 16692.696} C_VEL
LIN {X 0,Y 524.449,Z 1098.064,A -85,B 0,C 180,E1 16692.244,E2 16692.244} C_VEL
LIN {X 0,Y 515.777,Z 1113.842,A -85,B 0,C 180,E1 16691.257,E2 16691.257} C_VEL
LIN {X 0,Y 513.404,Z 1119.624,A -85,B 0,C 180,E1 16690.746,E2 16690.746} C_VEL
LIN {X 0,Y 508.31,Z 1138.086,A -85,B 0,C 180,E1 16688.723,E2 16688.723} C_VEL
LIN {X 0,Y 503.882,Z 1154.097,A -85,B 0,C 180,E1 16686.749,E2 16686.749} C_VEL
LIN {X 0,Y 499.786,Z 1169.036,A -85,B 0,C 180,E1 16684.688,E2 16684.688} C_VEL
LIN {X 0,Y 495.173,Z 1186.359,A -85,B 0,C 180,E1 16681.994,E2 16681.994} C_VEL
LIN {X 0,Y 491.205,Z 1201.531,A -85,B 0,C 180,E1 16679.247,E2 16679.247} C_VEL
LIN {X 0,Y 488.451,Z 1213.011,A -85,B 0,C 180,E1 16676.9,E2 16676.9} C_VEL
LIN {X 0,Y 486.068,Z 1223.768,A -85,B 0,C 180,E1 16674.426,E2 16674.426} C_VEL
LIN {X 0,Y 483.852,Z 1235.086,A -85,B 0,C 180,E1 16671.458,E2 16671.458} C_VEL
LIN {X 0,Y 482.085,Z 1245.438,A -85,B 0,C 180,E1 16668.206,E2 16668.206} C_VEL
LIN {X 0,Y 481.191,Z 1252.317,A -85,B 0,C 180,E1 16665.675,E2 16665.675} C_VEL
LIN {X 0,Y 480.561,Z 1258.205,A -85,B 0,C 180,E1 16663.111,E2 16663.111} C_VEL
LIN {X 0,Y 480.204,Z 1263.012,A -85,B 0,C 180,E1 16660.561,E2 16660.561} C_VEL
LIN {X 0,Y 479.974,Z 1267.079,A -85,B 0,C 180,E1 16657.785,E2 16657.785} C_VEL
LIN {X 0,Y 479.919,Z 1270.237,A -85,B 0,C 180,E1 16654.664,E2 16654.664} C_VEL
LIN {X 0,Y 479.906,Z 1271.68,A -85,B 0,C 180,E1 16651.675,E2 16651.675} C_VEL
LIN {X 0,Y 479.866,Z 1271.857,A -85,B 0,C 180,E1 16649.168,E2 16649.168} C_VEL
LIN {X 0,Y 479.912,Z 1271.041,A -85,B 0,C 180,E1 16646.659,E2 16646.659} C_VEL
LIN {X 0,Y 479.941,Z 1269.234,A -85,B 0,C 180,E1 16644.145,E2 16644.145} C_VEL
LIN {X 0,Y 480.019,Z 1266.411,A -85,B 0,C 180,E1 16641.62,E2 16641.62} C_VEL
LIN {X 0,Y 480.234,Z 1262.35,A -85,B 0,C 180,E1 16638.961,E2 16638.961} C_VEL
LIN {X 0,Y 480.666,Z 1257.123,A -85,B 0,C 180,E1 16636.28,E2 16636.28} C_VEL
LIN {X 0,Y 481.641,Z 1248.759,A -85,B 0,C 180,E1 16632.859,E2 16632.859} C_VEL
LIN {X 0,Y 482.885,Z 1240.291,A -85,B 0,C 180,E1 16630.027,E2 16630.027} C_VEL
LIN {X 0,Y 484.425,Z 1231.789,A -85,B 0,C 180,E1 16627.556,E2 16627.556} C_VEL
LIN {X 0,Y 486.473,Z 1221.833,A -85,B 0,C 180,E1 16625.017,E2 16625.017} C_VEL
LIN {X 0,Y 489.599,Z 1208.293,A -85,B 0,C 180,E1 16621.989,E2 16621.989} C_VEL
LIN {X 0,Y 493.297,Z 1193.387,A -85,B 0,C 180,E1 16619.154,E2 16619.154} C_VEL
LIN {X 0,Y 496.705,Z 1180.319,A -85,B 0,C 180,E1 16616.945,E2 16616.945} C_VEL
LIN {X 0,Y 500.424,Z 1166.641,A -85,B 0,C 180,E1 16614.875,E2 16614.875} C_VEL
LIN {X 0,Y 504.997,Z 1150.129,A -85,B 0,C 180,E1 16612.643,E2 16612.643} C_VEL
LIN {X 0,Y 510.741,Z 1129.355,A -85,B 0,C 180,E1 16610.202,E2 16610.202} C_VEL
LIN {X 0,Y 515.384,Z 1112.236,A -85,B 0,C 180,E1 16608.439,E2 16608.439} C_VEL
LIN {X 0,Y 519.884,Z 1095.187,A -85,B 0,C 180,E1 16606.871,E2 16606.871} C_VEL
LIN {X 0,Y 524.517,Z 1076.983,A -85,B 0,C 180,E1 16605.381,E2 16605.381} C_VEL
LIN {X 0,Y 529.859,Z 1055.026,A -85,B 0,C 180,E1 16603.803,E2 16603.803} C_VEL
LIN {X 0,Y 535.29,Z 1030.413,A -85,B 0,C 180,E1 16602.301,E2 16602.301} C_VEL
LIN {X 0,Y 539.496,Z 1009.433,A -85,B 0,C 180,E1 16601.203,E2 16601.203} C_VEL
LIN {X 0,Y 543,Z 990.282,A -85,B 0,C 180,E1 16600.336,E2 16600.336} C_VEL
LIN {X 0,Y 546.366,Z 969.716,A -85,B 0,C 180,E1 16599.539,E2 16599.539} C_VEL
LIN {X 0,Y 549.533,Z 947.412,A -85,B 0,C 180,E1 16598.815,E2 16598.815} C_VEL
LIN {X 0,Y 552.821,Z 918.612,A -85,B 0,C 180,E1 16598.084,E2 16598.084} C_VEL
LIN {X 0,Y 554.785,Z 894.704,A -85,B 0,C 180,E1 16597.637,E2 16597.637} C_VEL
LIN {X 0,Y 564.194,Z 690.947,A -85,B 0,C 180,E1 16594.562,E2 16594.562} C_VEL
LIN {X 0,Y 571.325,Z 540.391,A -85,B 0,C 180,E1 16592.262,E2 16592.262} C_VEL
LIN {X 0,Y 559.652,Z 522.767,A -85,B 0,C 180,E1 16589.869,E2 16589.869} C_VEL
LIN {X 0,Y 549.578,Z 509.317,A -85,B 0,C 180,E1 16587.612,E2 16587.612} C_VEL
LIN {X 0,Y 541.161,Z 498.545,A -85,B 0,C 180,E1 16585.529,E2 16585.529} C_VEL
LIN {X 0,Y 536.813,Z 493.175,A -85,B 0,C 180,E1 16584.367,E2 16584.367} C_VEL
LIN {X 0,Y 532.75,Z 488.141,A -85,B 0,C 180,E1 16583.212,E2 16583.212} C_VEL
LIN {X 0,Y 528.211,Z 482.669,A -85,B 0,C 180,E1 16581.837,E2 16581.837} C_VEL
LIN {X 0,Y 524.383,Z 478.107,A -85,B 0,C 180,E1 16580.592,E2 16580.592} C_VEL
LIN {X 0,Y 523.015,Z 476.576,A -85,B 0,C 180,E1 16580.128,E2 16580.128} C_VEL
LIN {X 0,Y 519.494,Z 472.485,A -85,B 0,C 180,E1 16578.866,E2 16578.866} C_VEL
LIN {X 0,Y 518.396,Z 470.957,A -85,B 0,C 180,E1 16578.441,E2 16578.441} C_VEL
LIN {X 0,Y 514.975,Z 467.681,A -85,B 0,C 180,E1 16577.107,E2 16577.107} C_VEL
LIN {X 0,Y 513.161,Z 464.836,A -85,B 0,C 180,E1 16576.295,E2 16576.295} C_VEL
LIN {X 0,Y 509.766,Z 461.951,A -85,B 0,C 180,E1 16574.773,E2 16574.773} C_VEL
LIN {X 0,Y 507.514,Z 458.334,A -85,B 0,C 180,E1 16573.559,E2 16573.559} C_VEL
LIN {X 0,Y 504.096,Z 456.007,A -85,B 0,C 180,E1 16571.673,E2 16571.673} C_VEL
LIN {X 0,Y 502.006,Z 452.245,A -85,B 0,C 180,E1 16570.153,E2 16570.153} C_VEL
LIN {X 0,Y 501.472,Z 451.68,A -85,B 0,C 180,E1 16569.758,E2 16569.758} C_VEL
LIN {X 0,Y 497.505,Z 449.084,A -85,B 0,C 180,E1 16566.231,E2 16566.231} C_VEL
LIN {X 0,Y 495.875,Z 445.291,A -85,B 0,C 180,E1 16563.295,E2 16563.295} C_VEL
LIN {X 0,Y 495.434,Z 444.954,A -85,B 0,C 180,E1 16562.082,E2 16562.082} C_VEL
LIN {X 0,Y 495.853,Z 445.214,A -85,B 0,C 180,E1 16556.879,E2 16556.879} C_VEL
LIN {X 0,Y 497.69,Z 449.309,A -85,B 0,C 180,E1 16553.656,E2 16553.656} C_VEL
LIN {X 0,Y 501.626,Z 451.73,A -85,B 0,C 180,E1 16550.245,E2 16550.245} C_VEL
LIN {X 0,Y 502.066,Z 452.388,A -85,B 0,C 180,E1 16549.906,E2 16549.906} C_VEL
LIN {X 0,Y 504.082,Z 456.016,A -85,B 0,C 180,E1 16548.443,E2 16548.443} C_VEL
LIN {X 0,Y 507.498,Z 458.353,A -85,B 0,C 180,E1 16546.556,E2 16546.556} C_VEL
LIN {X 0,Y 510.775,Z 463.098,A -85,B 0,C 180,E1 16544.85,E2 16544.85} C_VEL
LIN {X 0,Y 513.51,Z 465.3,A -85,B 0,C 180,E1 16543.658,E2 16543.658} C_VEL
LIN {X 0,Y 516.261,Z 469.248,A -85,B 0,C 180,E1 16542.472,E2 16542.472} C_VEL
LIN {X 0,Y 519.004,Z 471.698,A -85,B 0,C 180,E1 16541.436,E2 16541.436} C_VEL
LIN {X 0,Y 522.375,Z 476.015,A -85,B 0,C 180,E1 16540.196,E2 16540.196} C_VEL
LIN {X 0,Y 524.228,Z 477.88,A -85,B 0,C 180,E1 16539.571,E2 16539.571} C_VEL
LIN {X 0,Y 528.018,Z 482.516,A -85,B 0,C 180,E1 16538.33,E2 16538.33} C_VEL
LIN {X 0,Y 529.747,Z 484.599,A -85,B 0,C 180,E1 16537.792,E2 16537.792} C_VEL
LIN {X 0,Y 534.642,Z 490.52,A -85,B 0,C 180,E1 16536.349,E2 16536.349} C_VEL
LIN {X 0,Y 541.255,Z 499.37,A -85,B 0,C 180,E1 16534.534,E2 16534.534} C_VEL
LIN {X 0,Y 548.413,Z 509.129,A -85,B 0,C 180,E1 16532.736,E2 16532.736} C_VEL
LIN {X 0,Y 557.661,Z 522.429,A -85,B 0,C 180,E1 16530.607,E2 16530.607} C_VEL
LIN {X 0,Y 567.961,Z 538.031,A -85,B 0,C 180,E1 16528.446,E2 16528.446} C_VEL
LIN {X 0,Y 571.404,Z 543.913,A -85,B 0,C 180,E1 16527.753,E2 16527.753} C_VEL
LIN {X 0,Y 561.123,Z 761.25,A -85,B 0,C 180,E1 16524.462,E2 16524.462} C_VEL
LIN {X 0,Y 554.608,Z 902.829,A -85,B 0,C 180,E1 16522.324,E2 16522.324} C_VEL
LIN {X 0,Y 552.401,Z 929.105,A -85,B 0,C 180,E1 16521.828,E2 16521.828} C_VEL
LIN {X 0,Y 549.136,Z 956.401,A -85,B 0,C 180,E1 16521.123,E2 16521.123} C_VEL
LIN {X 0,Y 546.059,Z 977.853,A -85,B 0,C 180,E1 16520.426,E2 16520.426} C_VEL
LIN {X 0,Y 542.651,Z 998.551,A -85,B 0,C 180,E1 16519.625,E2 16519.625} C_VEL
LIN {X 0,Y 538.78,Z 1019.576,A -85,B 0,C 180,E1 16518.671,E2 16518.671} C_VEL
LIN {X 0,Y 533.686,Z 1044.665,A -85,B 0,C 180,E1 16517.331,E2 16517.331} C_VEL
LIN {X 0,Y 528.425,Z 1067.713,A -85,B 0,C 180,E1 16515.866,E2 16515.866} C_VEL
LIN {X 0,Y 523.782,Z 1086.932,A -85,B 0,C 180,E1 16514.468,E2 16514.468} C_VEL
LIN {X 0,Y 519.123,Z 1105.36,A -85,B 0,C 180,E1 16512.952,E2 16512.952} C_VEL
LIN {X 0,Y 513.435,Z 1127.13,A -85,B 0,C 180,E1 16510.921,E2 16510.921} C_VEL
LIN {X 0,Y 507.972,Z 1147.133,A -85,B 0,C 180,E1 16508.746,E2 16508.746} C_VEL
LIN {X 0,Y 503.706,Z 1162.807,A -85,B 0,C 180,E1 16506.827,E2 16506.827} C_VEL
LIN {X 0,Y 499.646,Z 1177.875,A -85,B 0,C 180,E1 16504.768,E2 16504.768} C_VEL
LIN {X 0,Y 495.278,Z 1194.601,A -85,B 0,C 180,E1 16502.201,E2 16502.201} C_VEL
LIN {X 0,Y 491.201,Z 1210.514,A -85,B 0,C 180,E1 16499.373,E2 16499.373} C_VEL
LIN {X 0,Y 488.332,Z 1222.763,A -85,B 0,C 180,E1 16496.9,E2 16496.9} C_VEL
LIN {X 0,Y 485.983,Z 1233.652,A -85,B 0,C 180,E1 16494.423,E2 16494.423} C_VEL
LIN {X 0,Y 483.733,Z 1245.58,A -85,B 0,C 180,E1 16491.329,E2 16491.329} C_VEL
LIN {X 0,Y 482.088,Z 1255.452,A -85,B 0,C 180,E1 16488.247,E2 16488.247} C_VEL
LIN {X 0,Y 481.176,Z 1262.447,A -85,B 0,C 180,E1 16485.668,E2 16485.668} C_VEL
LIN {X 0,Y 480.553,Z 1268.314,A -85,B 0,C 180,E1 16483.104,E2 16483.104} C_VEL
LIN {X 0,Y 480.197,Z 1273.1,A -85,B 0,C 180,E1 16480.554,E2 16480.554} C_VEL
LIN {X 0,Y 479.973,Z 1277.31,A -85,B 0,C 180,E1 16477.658,E2 16477.658} C_VEL
LIN {X 0,Y 479.92,Z 1280.335,A -85,B 0,C 180,E1 16474.537,E2 16474.537} C_VEL
LIN {X 0,Y 479.907,Z 1281.69,A -85,B 0,C 180,E1 16471.668,E2 16471.668} C_VEL
LIN {X 0,Y 479.867,Z 1281.847,A -85,B 0,C 180,E1 16469.161,E2 16469.161} C_VEL
LIN {X 0,Y 479.912,Z 1281.011,A -85,B 0,C 180,E1 16466.652,E2 16466.652} C_VEL
LIN {X 0,Y 479.941,Z 1279.184,A -85,B 0,C 180,E1 16464.138,E2 16464.138} C_VEL
LIN {X 0,Y 480.015,Z 1276.416,A -85,B 0,C 180,E1 16461.67,E2 16461.67} C_VEL
LIN {X 0,Y 480.231,Z 1272.469,A -85,B 0,C 180,E1 16459.075,E2 16459.075} C_VEL
LIN {X 0,Y 480.634,Z 1267.536,A -85,B 0,C 180,E1 16456.523,E2 16456.523} C_VEL
LIN {X 0,Y 481.485,Z 1260.001,A -85,B 0,C 180,E1 16453.344,E2 16453.344} C_VEL
LIN {X 0,Y 482.775,Z 1250.87,A -85,B 0,C 180,E1 16450.267,E2 16450.267} C_VEL
LIN {X 0,Y 484.274,Z 1242.328,A -85,B 0,C 180,E1 16447.797,E2 16447.797} C_VEL
LIN {X 0,Y 486.201,Z 1232.592,A -85,B 0,C 180,E1 16445.322,E2 16445.322} C_VEL
LIN {X 0,Y 488.612,Z 1221.582,A -85,B 0,C 180,E1 16442.846,E2 16442.846} C_VEL
LIN {X 0,Y 492.124,Z 1206.969,A -85,B 0,C 180,E1 16439.945,E2 16439.945} C_VEL
LIN {X 0,Y 496.238,Z 1190.682,A -85,B 0,C 180,E1 16437.177,E2 16437.177} C_VEL
LIN {X 0,Y 499.898,Z 1176.908,A -85,B 0,C 180,E1 16435.093,E2 16435.093} C_VEL
LIN {X 0,Y 503.974,Z 1161.824,A -85,B 0,C 180,E1 16433.045,E2 16433.045} C_VEL
LIN {X 0,Y 508.998,Z 1143.477,A -85,B 0,C 180,E1 16430.828,E2 16430.828} C_VEL
LIN {X 0,Y 514.594,Z 1122.664,A -85,B 0,C 180,E1 16428.649,E2 16428.649} C_VEL
LIN {X 0,Y 519.298,Z 1104.646,A -85,B 0,C 180,E1 16426.989,E2 16426.989} C_VEL
LIN {X 0,Y 523.801,Z 1086.816,A -85,B 0,C 180,E1 16425.526,E2 16425.526} C_VEL
LIN {X 0,Y 528.415,Z 1067.699,A -85,B 0,C 180,E1 16424.135,E2 16424.135} C_VEL
LIN {X 0,Y 533.918,Z 1043.607,A -85,B 0,C 180,E1 16422.608,E2 16422.608} C_VEL
LIN {X 0,Y 538.938,Z 1018.66,A -85,B 0,C 180,E1 16421.287,E2 16421.287} C_VEL
LIN {X 0,Y 542.67,Z 998.331,A -85,B 0,C 180,E1 16420.368,E2 16420.368} C_VEL
LIN {X 0,Y 546.077,Z 977.593,A -85,B 0,C 180,E1 16419.567,E2 16419.567} C_VEL
LIN {X 0,Y 549.23,Z 955.55,A -85,B 0,C 180,E1 16418.854,E2 16418.854} C_VEL
LIN {X 0,Y 552.576,Z 926.842,A -85,B 0,C 180,E1 16418.127,E2 16418.127} C_VEL
LIN {X 0,Y 554.611,Z 902.288,A -85,B 0,C 180,E1 16417.669,E2 16417.669} C_VEL
LIN {X 0,Y 563.89,Z 700.186,A -85,B 0,C 180,E1 16414.62,E2 16414.62} C_VEL
LIN {X 0,Y 571.312,Z 543.464,A -85,B 0,C 180,E1 16412.233,E2 16412.233} C_VEL
LIN {X 0,Y 562.015,Z 529.074,A -85,B 0,C 180,E1 16410.349,E2 16410.349} C_VEL
LIN {X 0,Y 551.98,Z 514.128,A -85,B 0,C 180,E1 16408.128,E2 16408.128} C_VEL
LIN {X 0,Y 542.964,Z 501.702,A -85,B 0,C 180,E1 16405.936,E2 16405.936} C_VEL
LIN {X 0,Y 535.87,Z 492.122,A -85,B 0,C 180,E1 16404.032,E2 16404.032} C_VEL
LIN {X 0,Y 532.441,Z 487.858,A -85,B 0,C 180,E1 16403.051,E2 16403.051} C_VEL
LIN {X 0,Y 528.239,Z 482.714,A -85,B 0,C 180,E1 16401.778,E2 16401.778} C_VEL
LIN {X 0,Y 524.407,Z 478.188,A -85,B 0,C 180,E1 16400.538,E2 16400.538} C_VEL
LIN {X 0,Y 523.18,Z 476.72,A -85,B 0,C 180,E1 16400.122,E2 16400.122} C_VEL
LIN {X 0,Y 519.621,Z 472.71,A -85,B 0,C 180,E1 16398.861,E2 16398.861} C_VEL
LIN {X 0,Y 518.529,Z 471.046,A -85,B 0,C 180,E1 16398.436,E2 16398.436} C_VEL
LIN {X 0,Y 515.07,Z 467.822,A -85,B 0,C 180,E1 16397.104,E2 16397.104} C_VEL
LIN {X 0,Y 513.25,Z 464.874,A -85,B 0,C 180,E1 16396.292,E2 16396.292} C_VEL
LIN {X 0,Y 509.815,Z 462.025,A -85,B 0,C 180,E1 16394.772,E2 16394.772} C_VEL
LIN {X 0,Y 507.543,Z 458.343,A -85,B 0,C 180,E1 16393.558,E2 16393.558} C_VEL
LIN {X 0,Y 504.174,Z 456.085,A -85,B 0,C 180,E1 16391.729,E2 16391.729} C_VEL
LIN {X 0,Y 502.033,Z 452.347,A -85,B 0,C 180,E1 16390.21,E2 16390.21} C_VEL
LIN {X 0,Y 501.583,Z 451.704,A -85,B 0,C 180,E1 16389.872,E2 16389.872} C_VEL
LIN {X 0,Y 497.682,Z 449.256,A -85,B 0,C 180,E1 16386.576,E2 16386.576} C_VEL
LIN {X 0,Y 495.875,Z 445.363,A -85,B 0,C 180,E1 16383.7,E2 16383.7} C_VEL
LIN {X 0,Y 495.618,Z 444.963,A -85,B 0,C 180,E1 16383.123,E2 16383.123} C_VEL
LIN {X 0,Y 495.853,Z 445.165,A -85,B 0,C 180,E1 16376.184,E2 16376.184} C_VEL
LIN {X 0,Y 497.324,Z 448.762,A -85,B 0,C 180,E1 16373.651,E2 16373.651} C_VEL
LIN {X 0,Y 500.978,Z 451.502,A -85,B 0,C 180,E1 16370.349,E2 16370.349} C_VEL
LIN {X 0,Y 501.946,Z 452.014,A -85,B 0,C 180,E1 16369.672,E2 16369.672} C_VEL
LIN {X 0,Y 503.696,Z 455.497,A -85,B 0,C 180,E1 16368.376,E2 16368.376} C_VEL
LIN {X 0,Y 506.94,Z 458.09,A -85,B 0,C 180,E1 16366.541,E2 16366.541} C_VEL
LIN {X 0,Y 507.861,Z 458.747,A -85,B 0,C 180,E1 16366.073,E2 16366.073} C_VEL
LIN {X 0,Y 510.335,Z 462.639,A -85,B 0,C 180,E1 16364.779,E2 16364.779} C_VEL
LIN {X 0,Y 513.559,Z 465.355,A -85,B 0,C 180,E1 16363.369,E2 16363.369} C_VEL
LIN {X 0,Y 516.477,Z 469.387,A -85,B 0,C 180,E1 16362.13,E2 16362.13} C_VEL
LIN {X 0,Y 519.031,Z 471.655,A -85,B 0,C 180,E1 16361.175,E2 16361.175} C_VEL
LIN {X 0,Y 522.341,Z 475.941,A -85,B 0,C 180,E1 16359.961,E2 16359.961} C_VEL
LIN {X 0,Y 524.281,Z 477.896,A -85,B 0,C 180,E1 16359.31,E2 16359.31} C_VEL
LIN {X 0,Y 528.007,Z 482.46,A -85,B 0,C 180,E1 16358.095,E2 16358.095} C_VEL
LIN {X 0,Y 529.827,Z 484.639,A -85,B 0,C 180,E1 16357.532,E2 16357.532} C_VEL
LIN {X 0,Y 534.479,Z 490.249,A -85,B 0,C 180,E1 16356.166,E2 16356.166} C_VEL
LIN {X 0,Y 539.281,Z 496.239,A -85,B 0,C 180,E1 16354.846,E2 16354.846} C_VEL
LIN {X 0,Y 547.092,Z 506.033,A -85,B 0,C 180,E1 16352.871,E2 16352.871} C_VEL
LIN {X 0,Y 558.397,Z 521.059,A -85,B 0,C 180,E1 16350.293,E2 16350.293} C_VEL
LIN {X 0,Y 568.196,Z 535.606,A -85,B 0,C 180,E1 16348.253,E2 16348.253} C_VEL
LIN {X 0,Y 571.356,Z 540.675,A -85,B 0,C 180,E1 16347.625,E2 16347.625} C_VEL
LIN {X 0,Y 561.115,Z 756.831,A -85,B 0,C 180,E1 16344.352,E2 16344.352} C_VEL
LIN {X 0,Y 554.709,Z 895.504,A -85,B 0,C 180,E1 16342.257,E2 16342.257} C_VEL
LIN {X 0,Y 552.528,Z 921.71,A -85,B 0,C 180,E1 16341.758,E2 16341.758} C_VEL
LIN {X 0,Y 549.303,Z 948.906,A -85,B 0,C 180,E1 16341.048,E2 16341.048} C_VEL
LIN {X 0,Y 546.312,Z 969.907,A -85,B 0,C 180,E1 16340.362,E2 16340.362} C_VEL
LIN {X 0,Y 543.045,Z 989.924,A -85,B 0,C 180,E1 16339.586,E2 16339.586} C_VEL
LIN {X 0,Y 539.528,Z 1009.173,A -85,B 0,C 180,E1 16338.718,E2 16338.718} C_VEL
LIN {X 0,Y 535.546,Z 1029.121,A -85,B 0,C 180,E1 16337.678,E2 16337.678} C_VEL
LIN {X 0,Y 530.902,Z 1050.448,A -85,B 0,C 180,E1 16336.401,E2 16336.401} C_VEL
LIN {X 0,Y 524.945,Z 1075.274,A -85,B 0,C 180,E1 16334.658,E2 16334.658} C_VEL
LIN {X 0,Y 520.284,Z 1093.626,A -85,B 0,C 180,E1 16333.172,E2 16333.172} C_VEL
LIN {X 0,Y 515.923,Z 1110.204,A -85,B 0,C 180,E1 16331.665,E2 16331.665} C_VEL
LIN {X 0,Y 513.404,Z 1119.624,A -85,B 0,C 180,E1 16330.746,E2 16330.746} C_VEL
LIN {X 0,Y 511.011,Z 1125.408,A -85,B 0,C 180,E1 16330.215,E2 16330.215} C_VEL
LIN {X 0,Y 502.111,Z 1140.065,A -85,B 0,C 180,E1 16329.024,E2 16329.024} C_VEL
LIN {X 0,Y 499.787,Z 1145.411,A -85,B 0,C 180,E1 16328.454,E2 16328.454} C_VEL
LIN {X 0,Y 494.259,Z 1164.467,A -85,B 0,C 180,E1 16325.923,E2 16325.923} C_VEL
LIN {X 0,Y 490.058,Z 1179.104,A -85,B 0,C 180,E1 16323.711,E2 16323.711} C_VEL
LIN {X 0,Y 486.363,Z 1192.491,A -85,B 0,C 180,E1 16321.44,E2 16321.44} C_VEL
LIN {X 0,Y 482.961,Z 1205.411,A -85,B 0,C 180,E1 16318.979,E2 16318.979} C_VEL
LIN {X 0,Y 479.255,Z 1220.487,A -85,B 0,C 180,E1 16315.67,E2 16315.67} C_VEL
LIN {X 0,Y 476.902,Z 1231.086,A -85,B 0,C 180,E1 16312.955,E2 16312.955} C_VEL
LIN {X 0,Y 475.251,Z 1239.672,A -85,B 0,C 180,E1 16310.444,E2 16310.444} C_VEL
LIN {X 0,Y 473.939,Z 1247.489,A -85,B 0,C 180,E1 16307.816,E2 16307.816} C_VEL
LIN {X 0,Y 472.971,Z 1254.746,A -85,B 0,C 180,E1 16304.949,E2 16304.949} C_VEL
LIN {X 0,Y 472.326,Z 1261.564,A -85,B 0,C 180,E1 16301.605,E2 16301.605} C_VEL
LIN {X 0,Y 472.05,Z 1265.96,A -85,B 0,C 180,E1 16298.775,E2 16298.775} C_VEL
LIN {X 0,Y 471.953,Z 1268.912,A -85,B 0,C 180,E1 16296.206,E2 16296.206} C_VEL
LIN {X 0,Y 471.916,Z 1270.84,A -85,B 0,C 180,E1 16293.664,E2 16293.664} C_VEL
LIN {X 0,Y 471.892,Z 1271.771,A -85,B 0,C 180,E1 16291.218,E2 16291.218} C_VEL
LIN {X 0,Y 471.883,Z 1271.789,A -85,B 0,C 180,E1 16288.789,E2 16288.789} C_VEL
LIN {X 0,Y 471.914,Z 1270.893,A -85,B 0,C 180,E1 16286.339,E2 16286.339} C_VEL
LIN {X 0,Y 471.952,Z 1269.003,A -85,B 0,C 180,E1 16283.801,E2 16283.801} C_VEL
LIN {X 0,Y 472.051,Z 1266.087,A -85,B 0,C 180,E1 16281.232,E2 16281.232} C_VEL
LIN {X 0,Y 472.307,Z 1261.726,A -85,B 0,C 180,E1 16278.402,E2 16278.402} C_VEL
LIN {X 0,Y 472.943,Z 1254.98,A -85,B 0,C 180,E1 16275.057,E2 16275.057} C_VEL
LIN {X 0,Y 473.907,Z 1247.76,A -85,B 0,C 180,E1 16272.19,E2 16272.19} C_VEL
LIN {X 0,Y 475.192,Z 1239.977,A -85,B 0,C 180,E1 16269.561,E2 16269.561} C_VEL
LIN {X 0,Y 476.831,Z 1231.422,A -85,B 0,C 180,E1 16267.048,E2 16267.048} C_VEL
LIN {X 0,Y 478.974,Z 1221.679,A -85,B 0,C 180,E1 16264.535,E2 16264.535} C_VEL
LIN {X 0,Y 482.225,Z 1208.381,A -85,B 0,C 180,E1 16261.522,E2 16261.522} C_VEL
LIN {X 0,Y 486.101,Z 1193.474,A -85,B 0,C 180,E1 16258.646,E2 16258.646} C_VEL
LIN {X 0,Y 489.689,Z 1180.405,A -85,B 0,C 180,E1 16256.409,E2 16256.409} C_VEL
LIN {X 0,Y 493.591,Z 1166.728,A -85,B 0,C 180,E1 16254.315,E2 16254.315} C_VEL
LIN {X 0,Y 498.438,Z 1150.022,A -85,B 0,C 180,E1 16252.034,E2 16252.034} C_VEL
LIN {X 0,Y 504.445,Z 1129.164,A -85,B 0,C 180,E1 16249.566,E2 16249.566} C_VEL
LIN {X 0,Y 509.198,Z 1112.321,A -85,B 0,C 180,E1 16247.819,E2 16247.819} C_VEL
LIN {X 0,Y 513.877,Z 1095.271,A -85,B 0,C 180,E1 16246.24,E2 16246.24} C_VEL
LIN {X 0,Y 518.685,Z 1077.066,A -85,B 0,C 180,E1 16244.742,E2 16244.742} C_VEL
LIN {X 0,Y 524.004,Z 1055.917,A -85,B 0,C 180,E1 16243.212,E2 16243.212} C_VEL
LIN {X 0,Y 529.615,Z 1031.497,A -85,B 0,C 180,E1 16241.704,E2 16241.704} C_VEL
LIN {X 0,Y 533.948,Z 1010.641,A -85,B 0,C 180,E1 16240.601,E2 16240.601} C_VEL
LIN {X 0,Y 537.784,Z 990.361,A -85,B 0,C 180,E1 16239.678,E2 16239.678} C_VEL
LIN {X 0,Y 541.279,Z 969.646,A -85,B 0,C 180,E1 16238.873,E2 16238.873} C_VEL
LIN {X 0,Y 544.58,Z 947.055,A -85,B 0,C 180,E1 16238.141,E2 16238.141} C_VEL
LIN {X 0,Y 547.949,Z 918.184,A -85,B 0,C 180,E1 16237.413,E2 16237.413} C_VEL
LIN {X 0,Y 549.929,Z 894.649,A -85,B 0,C 180,E1 16236.973,E2 16236.973} C_VEL
LIN {X 0,Y 559.688,Z 690.772,A -85,B 0,C 180,E1 16233.881,E2 16233.881} C_VEL
LIN {X 0,Y 566.889,Z 544.923,A -85,B 0,C 180,E1 16231.651,E2 16231.651} C_VEL
LIN {X 0,Y 556.618,Z 529.199,A -85,B 0,C 180,E1 16229.486,E2 16229.486} C_VEL
LIN {X 0,Y 546.785,Z 515.962,A -85,B 0,C 180,E1 16227.234,E2 16227.234} C_VEL
LIN {X 0,Y 538.496,Z 505.248,A -85,B 0,C 180,E1 16225.135,E2 16225.135} C_VEL
LIN {X 0,Y 534.399,Z 500.127,A -85,B 0,C 180,E1 16224.014,E2 16224.014} C_VEL
LIN {X 0,Y 530.57,Z 495.333,A -85,B 0,C 180,E1 16222.902,E2 16222.902} C_VEL
LIN {X 0,Y 526.094,Z 489.913,A -85,B 0,C 180,E1 16221.519,E2 16221.519} C_VEL
LIN {X 0,Y 522.212,Z 485.034,A -85,B 0,C 180,E1 16220.219,E2 16220.219} C_VEL
LIN {X 0,Y 517.947,Z 480.271,A -85,B 0,C 180,E1 16218.691,E2 16218.691} C_VEL
LIN {X 0,Y 516.582,Z 478.468,A -85,B 0,C 180,E1 16218.158,E2 16218.158} C_VEL
LIN {X 0,Y 513.114,Z 474.871,A -85,B 0,C 180,E1 16216.762,E2 16216.762} C_VEL
LIN {X 0,Y 511.693,Z 472.572,A -85,B 0,C 180,E1 16216.11,E2 16216.11} C_VEL
LIN {X 0,Y 508.238,Z 469.504,A -85,B 0,C 180,E1 16214.527,E2 16214.527} C_VEL
LIN {X 0,Y 506.12,Z 466.123,A -85,B 0,C 180,E1 16213.365,E2 16213.365} C_VEL
LIN {X 0,Y 502.77,Z 463.705,A -85,B 0,C 180,E1 16211.471,E2 16211.471} C_VEL
LIN {X 0,Y 500.661,Z 459.794,A -85,B 0,C 180,E1 16209.89,E2 16209.89} C_VEL
LIN {X 0,Y 496.257,Z 456.729,A -85,B 0,C 180,E1 16205.898,E2 16205.898} C_VEL
LIN {X 0,Y 494.823,Z 452.984,A -85,B 0,C 180,E1 16203.07,E2 16203.07} C_VEL
LIN {X 0,Y 494.829,Z 453.125,A -85,B 0,C 180,E1 16196.988,E2 16196.988} C_VEL
LIN {X 0,Y 496.816,Z 457.391,A -85,B 0,C 180,E1 16193.529,E2 16193.529} C_VEL
LIN {X 0,Y 500.719,Z 459.934,A -85,B 0,C 180,E1 16190.169,E2 16190.169} C_VEL
LIN {X 0,Y 502.757,Z 463.713,A -85,B 0,C 180,E1 16188.645,E2 16188.645} C_VEL
LIN {X 0,Y 506.104,Z 466.139,A -85,B 0,C 180,E1 16186.751,E2 16186.751} C_VEL
LIN {X 0,Y 509.575,Z 471.016,A -85,B 0,C 180,E1 16184.93,E2 16184.93} C_VEL
LIN {X 0,Y 511.971,Z 473.005,A -85,B 0,C 180,E1 16183.87,E2 16183.87} C_VEL
LIN {X 0,Y 514.893,Z 477.072,A -85,B 0,C 180,E1 16182.599,E2 16182.599} C_VEL
LIN {X 0,Y 517.325,Z 479.296,A -85,B 0,C 180,E1 16181.665,E2 16181.665} C_VEL
LIN {X 0,Y 520.809,Z 483.705,A -85,B 0,C 180,E1 16180.368,E2 16180.368} C_VEL
LIN {X 0,Y 522.555,Z 485.606,A -85,B 0,C 180,E1 16179.766,E2 16179.766} C_VEL
LIN {X 0,Y 526.569,Z 490.358,A -85,B 0,C 180,E1 16178.443,E2 16178.443} C_VEL
LIN {X 0,Y 532.697,Z 498.02,A -85,B 0,C 180,E1 16176.58,E2 16176.58} C_VEL
LIN {X 0,Y 539.053,Z 506.653,A -85,B 0,C 180,E1 16174.805,E2 16174.805} C_VEL
LIN {X 0,Y 546.128,Z 516.447,A -85,B 0,C 180,E1 16172.996,E2 16172.996} C_VEL
LIN {X 0,Y 554.975,Z 529.339,A -85,B 0,C 180,E1 16170.922,E2 16170.922} C_VEL
LIN {X 0,Y 564.925,Z 544.598,A -85,B 0,C 180,E1 16168.791,E2 16168.791} C_VEL
LIN {X 0,Y 566.929,Z 548.177,A -85,B 0,C 180,E1 16168.375,E2 16168.375} C_VEL
LIN {X 0,Y 556.307,Z 765.031,A -85,B 0,C 180,E1 16165.078,E2 16165.078} C_VEL
LIN {X 0,Y 549.728,Z 902.837,A -85,B 0,C 180,E1 16162.986,E2 16162.986} C_VEL
LIN {X 0,Y 547.405,Z 929.681,A -85,B 0,C 180,E1 16162.477,E2 16162.477} C_VEL
LIN {X 0,Y 544.057,Z 956.647,A -85,B 0,C 180,E1 16161.775,E2 16161.775} C_VEL
LIN {X 0,Y 540.931,Z 977.772,A -85,B 0,C 180,E1 16161.088,E2 16161.088} C_VEL
LIN {X 0,Y 537.417,Z 998.468,A -85,B 0,C 180,E1 16160.286,E2 16160.286} C_VEL
LIN {X 0,Y 533.564,Z 1018.76,A -85,B 0,C 180,E1 16159.365,E2 16159.365} C_VEL
LIN {X 0,Y 528.378,Z 1043.667,A -85,B 0,C 180,E1 16158.04,E2 16158.04} C_VEL
LIN {X 0,Y 522.778,Z 1067.379,A -85,B 0,C 180,E1 16156.532,E2 16156.532} C_VEL
LIN {X 0,Y 518.101,Z 1086.108,A -85,B 0,C 180,E1 16155.166,E2 16155.166} C_VEL
LIN {X 0,Y 513.499,Z 1103.673,A -85,B 0,C 180,E1 16153.723,E2 16153.723} C_VEL
LIN {X 0,Y 508.835,Z 1120.827,A -85,B 0,C 180,E1 16152.143,E2 16152.143} C_VEL
LIN {X 0,Y 503.277,Z 1140.853,A -85,B 0,C 180,E1 16150.062,E2 16150.062} C_VEL
LIN {X 0,Y 497.503,Z 1160.953,A -85,B 0,C 180,E1 16147.639,E2 16147.639} C_VEL
LIN {X 0,Y 493.214,Z 1176.084,A -85,B 0,C 180,E1 16145.573,E2 16145.573} C_VEL
LIN {X 0,Y 489.367,Z 1189.859,A -85,B 0,C 180,E1 16143.476,E2 16143.476} C_VEL
LIN {X 0,Y 485.603,Z 1203.987,A -85,B 0,C 180,E1 16141.066,E2 16141.066} C_VEL
